	Pump2_Data_Exchange_Active_CMD_Value.16	:= GracoSealer_Inputs.Byte52.0;
	Pump2_Data_Exchange_Active_CMD_Value.17	:= GracoSealer_Inputs.Byte52.1;
	Pump2_Data_Exchange_Active_CMD_Value.18	:= GracoSealer_Inputs.Byte52.2;
	Pump2_Data_Exchange_Active_CMD_Value.19	:= GracoSealer_Inputs.Byte52.3;
	Pump2_Data_Exchange_Active_CMD_Value.20	:= GracoSealer_Inputs.Byte52.4;
	Pump2_Data_Exchange_Active_CMD_Value.21	:= GracoSealer_Inputs.Byte52.5;
	Pump2_Data_Exchange_Active_CMD_Value.22	:= GracoSealer_Inputs.Byte52.6;
	Pump2_Data_Exchange_Active_CMD_Value.23	:= GracoSealer_Inputs.Byte52.7;

	Pump2_Data_Exchange_Active_CMD_Value.24	:= GracoSealer_Inputs.Byte53.0;
	Pump2_Data_Exchange_Active_CMD_Value.25	:= GracoSealer_Inputs.Byte53.1;
	Pump2_Data_Exchange_Active_CMD_Value.26	:= GracoSealer_Inputs.Byte53.2;
	Pump2_Data_Exchange_Active_CMD_Value.27	:= GracoSealer_Inputs.Byte53.3;
	Pump2_Data_Exchange_Active_CMD_Value.28	:= GracoSealer_Inputs.Byte53.4;
	Pump2_Data_Exchange_Active_CMD_Value.29	:= GracoSealer_Inputs.Byte53.5;
	Pump2_Data_Exchange_Active_CMD_Value.30	:= GracoSealer_Inputs.Byte53.6;
	Pump2_Data_Exchange_Active_CMD_Value.31	:= GracoSealer_Inputs.Byte53.7;



	(*Heat 1 - Inputs from Graco*)
	Heat1_Heartbeat								:= GracoSealer_Inputs.Byte54.0;
	Heat1_Enabled								:= GracoSealer_Inputs.Byte54.1;
	Heat1_Control_Active							:= GracoSealer_Inputs.Byte54.2;
	Heat1_ON									:= GracoSealer_Inputs.Byte54.3;
	Heat1_WarmingUp							:= GracoSealer_Inputs.Byte54.4;
	Heat1_At_Temp								:= GracoSealer_Inputs.Byte54.5;
	Heat1_Temp_Soak_Mode						:= GracoSealer_Inputs.Byte54.6;
	Heat1_SetBack_Mode							:= GracoSealer_Inputs.Byte54.7;


	Heat1_Off									:= GracoSealer_Inputs.Byte55.0;
	Heat1_Module_NoAlarms_Active				:= GracoSealer_Inputs.Byte55.1;
	Heat1_Module_NoDeviations_Active				:= GracoSealer_Inputs.Byte55.2;
	Heat1_Module_NoAdvisory_Active				:= GracoSealer_Inputs.Byte55.3;
	Heat1_Zone_NoAlarms_Active					:= GracoSealer_Inputs.Byte55.4;
	Heat1_Zone_NoDeviations_Active				:= GracoSealer_Inputs.Byte55.5;
	Heat1_Zone_NoAdvisory_Active				:= GracoSealer_Inputs.Byte55.6;
	Heat1_Idle_Timeout_Happened					:= GracoSealer_Inputs.Byte55.7;


	(*Byte 56 Reserved*)
	(*Byte 57 Reserved*)


	Heat1_Soak_Time_Remaining.0					:= GracoSealer_Inputs.Byte58.0;			(*xx seconds*)
	Heat1_Soak_Time_Remaining.1					:= GracoSealer_Inputs.Byte58.1;			(*xx seconds*)
	Heat1_Soak_Time_Remaining.2					:= GracoSealer_Inputs.Byte58.2;			(*xx seconds*)
	Heat1_Soak_Time_Remaining.3					:= GracoSealer_Inputs.Byte58.3;			(*xx seconds*)
	Heat1_Soak_Time_Remaining.4					:= GracoSealer_Inputs.Byte58.4;			(*xx seconds*)
	Heat1_Soak_Time_Remaining.5					:= GracoSealer_Inputs.Byte58.5;			(*xx seconds*)
	Heat1_Soak_Time_Remaining.6					:= GracoSealer_Inputs.Byte58.6;			(*xx seconds*)
	Heat1_Soak_Time_Remaining.7					:= GracoSealer_Inputs.Byte58.7;			(*xx seconds*)

	Heat1_Soak_Time_Remaining.8					:= GracoSealer_Inputs.Byte59.0;			(*xx seconds*)
	Heat1_Soak_Time_Remaining.9					:= GracoSealer_Inputs.Byte59.1;			(*xx seconds*)
	Heat1_Soak_Time_Remaining.10				:= GracoSealer_Inputs.Byte59.2;			(*xx seconds*)
	Heat1_Soak_Time_Remaining.11				:= GracoSealer_Inputs.Byte59.3;			(*xx seconds*)
	Heat1_Soak_Time_Remaining.12				:= GracoSealer_Inputs.Byte59.4;			(*xx seconds*)
	Heat1_Soak_Time_Remaining.13				:= GracoSealer_Inputs.Byte59.5;			(*xx seconds*)
	Heat1_Soak_Time_Remaining.14				:= GracoSealer_Inputs.Byte59.6;			(*xx seconds*)
	Heat1_Soak_Time_Remaining.15				:= GracoSealer_Inputs.Byte59.7;			(*xx seconds*)


	Heat1_Data_Exchange_Active_CMD.0			:= GracoSealer_Inputs.Byte60.0;
	Heat1_Data_Exchange_Active_CMD.1			:= GracoSealer_Inputs.Byte60.1;
	Heat1_Data_Exchange_Active_CMD.2			:= GracoSealer_Inputs.Byte60.2;
	Heat1_Data_Exchange_Active_CMD.3			:= GracoSealer_Inputs.Byte60.3;
	Heat1_Data_Exchange_Active_CMD.4			:= GracoSealer_Inputs.Byte60.4;
	Heat1_Data_Exchange_Active_CMD.5			:= GracoSealer_Inputs.Byte60.5;
	Heat1_Data_Exchange_Active_CMD.6			:= GracoSealer_Inputs.Byte60.6;
	Heat1_Data_Exchange_Active_CMD.7			:= GracoSealer_Inputs.Byte60.7;

	Heat1_Data_Exchange_Active_CMD.8			:= GracoSealer_Inputs.Byte61.0;
	Heat1_Data_Exchange_Active_CMD.9			:= GracoSealer_Inputs.Byte61.1;
	Heat1_Data_Exchange_Active_CMD.10			:= GracoSealer_Inputs.Byte61.2;
	Heat1_Data_Exchange_Active_CMD.11			:= GracoSealer_Inputs.Byte61.3;
	Heat1_Data_Exchange_Active_CMD.12			:= GracoSealer_Inputs.Byte61.4;
	Heat1_Data_Exchange_Active_CMD.13			:= GracoSealer_Inputs.Byte61.5;
	Heat1_Data_Exchange_Active_CMD.14			:= GracoSealer_Inputs.Byte61.6;
	Heat1_Data_Exchange_Active_CMD.15			:= GracoSealer_Inputs.Byte61.7;


	Heat1_Data_Exchange_Active_CMD_Value.0		:= GracoSealer_Inputs.Byte62.0;
	Heat1_Data_Exchange_Active_CMD_Value.1		:= GracoSealer_Inputs.Byte62.1;
	Heat1_Data_Exchange_Active_CMD_Value.2		:= GracoSealer_Inputs.Byte62.2;
	Heat1_Data_Exchange_Active_CMD_Value.3		:= GracoSealer_Inputs.Byte62.3;
	Heat1_Data_Exchange_Active_CMD_Value.4		:= GracoSealer_Inputs.Byte62.4;
	Heat1_Data_Exchange_Active_CMD_Value.5		:= GracoSealer_Inputs.Byte62.5;
	Heat1_Data_Exchange_Active_CMD_Value.6		:= GracoSealer_Inputs.Byte62.6;
	Heat1_Data_Exchange_Active_CMD_Value.7		:= GracoSealer_Inputs.Byte62.7;

	Heat1_Data_Exchange_Active_CMD_Value.8		:= GracoSealer_Inputs.Byte63.0;
	Heat1_Data_Exchange_Active_CMD_Value.9		:= GracoSealer_Inputs.Byte63.1;
	Heat1_Data_Exchange_Active_CMD_Value.10		:= GracoSealer_Inputs.Byte63.2;
	Heat1_Data_Exchange_Active_CMD_Value.11		:= GracoSealer_Inputs.Byte63.3;
	Heat1_Data_Exchange_Active_CMD_Value.12		:= GracoSealer_Inputs.Byte63.4;
	Heat1_Data_Exchange_Active_CMD_Value.13		:= GracoSealer_Inputs.Byte63.5;
	Heat1_Data_Exchange_Active_CMD_Value.14		:= GracoSealer_Inputs.Byte63.6;
	Heat1_Data_Exchange_Active_CMD_Value.15		:= GracoSealer_Inputs.Byte63.7;

	Heat1_Data_Exchange_Active_CMD_Value.16		:= GracoSealer_Inputs.Byte64.0;
	Heat1_Data_Exchange_Active_CMD_Value.17		:= GracoSealer_Inputs.Byte64.1;
	Heat1_Data_Exchange_Active_CMD_Value.18		:= GracoSealer_Inputs.Byte64.2;
	Heat1_Data_Exchange_Active_CMD_Value.19		:= GracoSealer_Inputs.Byte64.3;
	Heat1_Data_Exchange_Active_CMD_Value.20		:= GracoSealer_Inputs.Byte64.4;
	Heat1_Data_Exchange_Active_CMD_Value.21		:= GracoSealer_Inputs.Byte64.5;
	Heat1_Data_Exchange_Active_CMD_Value.22		:= GracoSealer_Inputs.Byte64.6;
	Heat1_Data_Exchange_Active_CMD_Value.23		:= GracoSealer_Inputs.Byte64.7;

	Heat1_Data_Exchange_Active_CMD_Value.24		:= GracoSealer_Inputs.Byte65.0;
	Heat1_Data_Exchange_Active_CMD_Value.25		:= GracoSealer_Inputs.Byte65.1;
	Heat1_Data_Exchange_Active_CMD_Value.26		:= GracoSealer_Inputs.Byte65.2;
	Heat1_Data_Exchange_Active_CMD_Value.27		:= GracoSealer_Inputs.Byte65.3;
	Heat1_Data_Exchange_Active_CMD_Value.28		:= GracoSealer_Inputs.Byte65.4;
	Heat1_Data_Exchange_Active_CMD_Value.29		:= GracoSealer_Inputs.Byte65.5;
	Heat1_Data_Exchange_Active_CMD_Value.30		:= GracoSealer_Inputs.Byte65.6;
	Heat1_Data_Exchange_Active_CMD_Value.31		:= GracoSealer_Inputs.Byte65.7;



	(*Heat 2 - Inputs from Graco. Only used if tandem pump is on*)
	Heat1_Heartbeat								:= GracoSealer_Inputs.Byte66.0;
	Heat2_Enabled								:= GracoSealer_Inputs.Byte66.1;
	Heat2_Control_Active							:= GracoSealer_Inputs.Byte66.2;
	Heat2_ON									:= GracoSealer_Inputs.Byte66.3;
	Heat2_WarmingUp							:= GracoSealer_Inputs.Byte66.4;
	Heat2_At_Temp								:= GracoSealer_Inputs.Byte66.5;
	Heat2_Temp_Soak_Mode						:= GracoSealer_Inputs.Byte66.6;
	Heat2_SetBack_Mode							:= GracoSealer_Inputs.Byte66.7;


	Heat2_Off									:= GracoSealer_Inputs.Byte67.0;
	Heat2_Module_NoAlarms_Active				:= GracoSealer_Inputs.Byte67.1;
	Heat2_Module_NoDeviations_Active				:= GracoSealer_Inputs.Byte67.2;
	Heat2_Module_NoAdvisory_Active				:= GracoSealer_Inputs.Byte67.3;
	Heat2_Zone_NoAlarms_Active					:= GracoSealer_Inputs.Byte67.4;
	Heat2_Zone_NoDeviations_Active				:= GracoSealer_Inputs.Byte67.5;
	Heat2_Zone_NoAdvisory_Active				:= GracoSealer_Inputs.Byte67.6;
	Heat2_Idle_Timeout_Happened					:= GracoSealer_Inputs.Byte67.7;


	(*Byte 68 Reserved*)
	(*Byte 69 Reserved*)


	Heat2_Soak_Time_Remaining.0					:= GracoSealer_Inputs.Byte70.0;			(*xx seconds*)
	Heat2_Soak_Time_Remaining.1					:= GracoSealer_Inputs.Byte70.1;			(*xx seconds*)
	Heat2_Soak_Time_Remaining.2					:= GracoSealer_Inputs.Byte70.2;			(*xx seconds*)
	Heat2_Soak_Time_Remaining.3					:= GracoSealer_Inputs.Byte70.3;			(*xx seconds*)
	Heat2_Soak_Time_Remaining.4					:= GracoSealer_Inputs.Byte70.4;			(*xx seconds*)
	Heat2_Soak_Time_Remaining.5					:= GracoSealer_Inputs.Byte70.5;			(*xx seconds*)
	Heat2_Soak_Time_Remaining.6					:= GracoSealer_Inputs.Byte70.6;			(*xx seconds*)
	Heat2_Soak_Time_Remaining.7					:= GracoSealer_Inputs.Byte70.7;			(*xx seconds*)

	Heat2_Soak_Time_Remaining.8					:= GracoSealer_Inputs.Byte71.0;			(*xx seconds*)
	Heat2_Soak_Time_Remaining.9					:= GracoSealer_Inputs.Byte71.1;			(*xx seconds*)
	Heat2_Soak_Time_Remaining.10				:= GracoSealer_Inputs.Byte71.2;			(*xx seconds*)
	Heat2_Soak_Time_Remaining.11				:= GracoSealer_Inputs.Byte71.3;			(*xx seconds*)
	Heat2_Soak_Time_Remaining.12				:= GracoSealer_Inputs.Byte71.4;			(*xx seconds*)
	Heat2_Soak_Time_Remaining.13				:= GracoSealer_Inputs.Byte71.5;			(*xx seconds*)
	Heat2_Soak_Time_Remaining.14				:= GracoSealer_Inputs.Byte71.6;			(*xx seconds*)
	Heat2_Soak_Time_Remaining.15				:= GracoSealer_Inputs.Byte71.7;			(*xx seconds*)


	Heat2_Data_Exchange_Active_CMD.0			:= GracoSealer_Inputs.Byte72.0;
	Heat2_Data_Exchange_Active_CMD.1			:= GracoSealer_Inputs.Byte72.1;
	Heat2_Data_Exchange_Active_CMD.2			:= GracoSealer_Inputs.Byte72.2;
	Heat2_Data_Exchange_Active_CMD.3			:= GracoSealer_Inputs.Byte72.3;
	Heat2_Data_Exchange_Active_CMD.4			:= GracoSealer_Inputs.Byte72.4;
	Heat2_Data_Exchange_Active_CMD.5			:= GracoSealer_Inputs.Byte72.5;
	Heat2_Data_Exchange_Active_CMD.6			:= GracoSealer_Inputs.Byte72.6;
	Heat2_Data_Exchange_Active_CMD.7			:= GracoSealer_Inputs.Byte72.7;

	Heat2_Data_Exchange_Active_CMD.8			:= GracoSealer_Inputs.Byte73.0;
	Heat2_Data_Exchange_Active_CMD.9			:= GracoSealer_Inputs.Byte73.1;
	Heat2_Data_Exchange_Active_CMD.10			:= GracoSealer_Inputs.Byte73.2;
	Heat2_Data_Exchange_Active_CMD.11			:= GracoSealer_Inputs.Byte73.3;
	Heat2_Data_Exchange_Active_CMD.12			:= GracoSealer_Inputs.Byte73.4;
	Heat2_Data_Exchange_Active_CMD.13			:= GracoSealer_Inputs.Byte73.5;
	Heat2_Data_Exchange_Active_CMD.14			:= GracoSealer_Inputs.Byte73.6;
	Heat2_Data_Exchange_Active_CMD.15			:= GracoSealer_Inputs.Byte73.7;


	Heat2_Data_Exchange_Active_CMD_Value.0		:= GracoSealer_Inputs.Byte74.0;
	Heat2_Data_Exchange_Active_CMD_Value.1		:= GracoSealer_Inputs.Byte74.1;
	Heat2_Data_Exchange_Active_CMD_Value.2		:= GracoSealer_Inputs.Byte74.2;
	Heat2_Data_Exchange_Active_CMD_Value.3		:= GracoSealer_Inputs.Byte74.3;
	Heat2_Data_Exchange_Active_CMD_Value.4		:= GracoSealer_Inputs.Byte74.4;
	Heat2_Data_Exchange_Active_CMD_Value.5		:= GracoSealer_Inputs.Byte74.5;
	Heat2_Data_Exchange_Active_CMD_Value.6		:= GracoSealer_Inputs.Byte74.6;
	Heat2_Data_Exchange_Active_CMD_Value.7		:= GracoSealer_Inputs.Byte74.7;

	Heat2_Data_Exchange_Active_CMD_Value.8		:= GracoSealer_Inputs.Byte75.0;
	Heat2_Data_Exchange_Active_CMD_Value.9		:= GracoSealer_Inputs.Byte75.1;
	Heat2_Data_Exchange_Active_CMD_Value.10		:= GracoSealer_Inputs.Byte75.2;
	Heat2_Data_Exchange_Active_CMD_Value.11		:= GracoSealer_Inputs.Byte75.3;
	Heat2_Data_Exchange_Active_CMD_Value.12		:= GracoSealer_Inputs.Byte75.4;
	Heat2_Data_Exchange_Active_CMD_Value.13		:= GracoSealer_Inputs.Byte75.5;
	Heat2_Data_Exchange_Active_CMD_Value.14		:= GracoSealer_Inputs.Byte75.6;
	Heat2_Data_Exchange_Active_CMD_Value.15		:= GracoSealer_Inputs.Byte75.7;

	Heat2_Data_Exchange_Active_CMD_Value.16		:= GracoSealer_Inputs.Byte76.0;
	Heat2_Data_Exchange_Active_CMD_Value.17		:= GracoSealer_Inputs.Byte76.1;
	Heat2_Data_Exchange_Active_CMD_Value.18		:= GracoSealer_Inputs.Byte76.2;
	Heat2_Data_Exchange_Active_CMD_Value.19		:= GracoSealer_Inputs.Byte76.3;
	Heat2_Data_Exchange_Active_CMD_Value.20		:= GracoSealer_Inputs.Byte76.4;
	Heat2_Data_Exchange_Active_CMD_Value.21		:= GracoSealer_Inputs.Byte76.5;
	Heat2_Data_Exchange_Active_CMD_Value.22		:= GracoSealer_Inputs.Byte76.6;
	Heat2_Data_Exchange_Active_CMD_Value.23		:= GracoSealer_Inputs.Byte76.7;

	Heat2_Data_Exchange_Active_CMD_Value.24		:= GracoSealer_Inputs.Byte77.0;
	Heat2_Data_Exchange_Active_CMD_Value.25		:= GracoSealer_Inputs.Byte77.1;
	Heat2_Data_Exchange_Active_CMD_Value.26		:= GracoSealer_Inputs.Byte77.2;
	Heat2_Data_Exchange_Active_CMD_Value.27		:= GracoSealer_Inputs.Byte77.3;
	Heat2_Data_Exchange_Active_CMD_Value.28		:= GracoSealer_Inputs.Byte77.4;
	Heat2_Data_Exchange_Active_CMD_Value.29		:= GracoSealer_Inputs.Byte77.5;
	Heat2_Data_Exchange_Active_CMD_Value.30		:= GracoSealer_Inputs.Byte77.6;
	Heat2_Data_Exchange_Active_CMD_Value.31		:= GracoSealer_Inputs.Byte77.7;







































(*end*)
END_ACTION

ACTION Outputs:



	GracoSealer_Outputs.Byte0.0	:= Pump1_Sys_Data_Exchange_CMD.0;
	GracoSealer_Outputs.Byte0.1	:= Pump1_Sys_Data_Exchange_CMD.1;
	GracoSealer_Outputs.Byte0.2	:= Pump1_Sys_Data_Exchange_CMD.2;
	GracoSealer_Outputs.Byte0.3	:= Pump1_Sys_Data_Exchange_CMD.3;
	GracoSealer_Outputs.Byte0.4	:= Pump1_Sys_Data_Exchange_CMD.4;
	GracoSealer_Outputs.Byte0.5	:= Pump1_Sys_Data_Exchange_CMD.5;
	GracoSealer_Outputs.Byte0.6	:= Pump1_Sys_Data_Exchange_CMD.6;
	GracoSealer_Outputs.Byte0.7	:= Pump1_Sys_Data_Exchange_CMD.7;

	GracoSealer_Outputs.Byte1.0	:= Pump1_Sys_Data_Exchange_CMD.8;
	GracoSealer_Outputs.Byte1.1	:= Pump1_Sys_Data_Exchange_CMD.9;
	GracoSealer_Outputs.Byte1.2	:= Pump1_Sys_Data_Exchange_CMD.10;
	GracoSealer_Outputs.Byte1.3	:= Pump1_Sys_Data_Exchange_CMD.11;
	GracoSealer_Outputs.Byte1.4	:= Pump1_Sys_Data_Exchange_CMD.12;
	GracoSealer_Outputs.Byte1.5	:= Pump1_Sys_Data_Exchange_CMD.13;
	GracoSealer_Outputs.Byte1.6	:= Pump1_Sys_Data_Exchange_CMD.14;
	GracoSealer_Outputs.Byte1.7	:= Pump1_Sys_Data_Exchange_CMD.15;


	GracoSealer_Outputs.Byte2.0	:= Pump1_Sys_Enable;
	GracoSealer_Outputs.Byte2.1	:= Pump1_Sys_Disable_REQ;
	GracoSealer_Outputs.Byte2.2	:= Pump1_Lockout;
	GracoSealer_Outputs.Byte2.3	:= Pump1_Style_Enable;
	GracoSealer_Outputs.Byte2.4	:= Pump1_Go;
	GracoSealer_Outputs.Byte2.5	:= Pump1_Disp_Complete;
	GracoSealer_Outputs.Byte2.6	:= Pump1_Tandem_Cross_REQ;
	GracoSealer_Outputs.Byte2.7	:= Pump2_Prime_Inactive_Pump_REQ;


	GracoSealer_Outputs.Byte3.0	:= Pump1_Valve_Depressurization_REQ;
	GracoSealer_Outputs.Byte3.1	:= Pump1_Platen_Depressurization_REQ;
	GracoSealer_Outputs.Byte3.2	:= Pump1_Auto_Depressurization_Cancel_REQ;
	GracoSealer_Outputs.Byte3.3	:= Pump_Acknowledge_Clear_Errors;
	(*Byte3.4 Reserved Bit 1*)
	(*Byte3.5 Reserved Bit 2*)
	(*Byte 3.6 Reserved Bit 3*)
	(*Byte 3.7 Reserved Bit 4*)


	GracoSealer_Outputs.Byte4.0	:= Pump1_Desired_Style_Numb.0;
	GracoSealer_Outputs.Byte4.1	:= Pump1_Desired_Style_Numb.1;
	GracoSealer_Outputs.Byte4.2	:= Pump1_Desired_Style_Numb.2;
	GracoSealer_Outputs.Byte4.3	:= Pump1_Desired_Style_Numb.3;
	GracoSealer_Outputs.Byte4.4	:= Pump1_Desired_Style_Numb.4;
	GracoSealer_Outputs.Byte4.5	:= Pump1_Desired_Style_Numb.5;
	GracoSealer_Outputs.Byte4.6	:= Pump1_Desired_Style_Numb.6;
	GracoSealer_Outputs.Byte4.7	:= Pump1_Desired_Style_Numb.7;

	GracoSealer_Outputs.Byte5.0	:= Pump1_Desired_Style_Numb.8;
	GracoSealer_Outputs.Byte5.1	:= Pump1_Desired_Style_Numb.9;
	GracoSealer_Outputs.Byte5.2	:= Pump1_Desired_Style_Numb.10;
	GracoSealer_Outputs.Byte5.3	:= Pump1_Desired_Style_Numb.11;
	GracoSealer_Outputs.Byte5.4	:= Pump1_Desired_Style_Numb.12;
	GracoSealer_Outputs.Byte5.5	:= Pump1_Desired_Style_Numb.13;
	GracoSealer_Outputs.Byte5.6	:= Pump1_Desired_Style_Numb.14;
	GracoSealer_Outputs.Byte5.7	:= Pump1_Desired_Style_Numb.15;


	GracoSealer_Outputs.Byte6.0	:= Pump1_Style_PreCharge_REQ.0;		(*xxx.x bars*)
	GracoSealer_Outputs.Byte6.1	:= Pump1_Style_PreCharge_REQ.1;		(*xxx.x bars*)
	GracoSealer_Outputs.Byte6.2	:= Pump1_Style_PreCharge_REQ.2;		(*xxx.x bars*)
	GracoSealer_Outputs.Byte6.3	:= Pump1_Style_PreCharge_REQ.3;		(*xxx.x bars*)
	GracoSealer_Outputs.Byte6.4	:= Pump1_Style_PreCharge_REQ.4;		(*xxx.x bars*)
	GracoSealer_Outputs.Byte6.5	:= Pump1_Style_PreCharge_REQ.5;		(*xxx.x bars*)
	GracoSealer_Outputs.Byte6.6	:= Pump1_Style_PreCharge_REQ.6;		(*xxx.x bars*)
	GracoSealer_Outputs.Byte6.7	:= Pump1_Style_PreCharge_REQ.7;		(*xxx.x bars*)

	GracoSealer_Outputs.Byte7.0	:= Pump1_Style_PreCharge_REQ.8;		(*xxx.x bars*)
	GracoSealer_Outputs.Byte7.1	:= Pump1_Style_PreCharge_REQ.9;		(*xxx.x bars*)
	GracoSealer_Outputs.Byte7.2	:= Pump1_Style_PreCharge_REQ.10;		(*xxx.x bars*)
	GracoSealer_Outputs.Byte7.3	:= Pump1_Style_PreCharge_REQ.11;		(*xxx.x bars*)
	GracoSealer_Outputs.Byte7.4	:= Pump1_Style_PreCharge_REQ.12;		(*xxx.x bars*)
	GracoSealer_Outputs.Byte7.5	:= Pump1_Style_PreCharge_REQ.13;		(*xxx.x bars*)
	GracoSealer_Outputs.Byte7.6	:= Pump1_Style_PreCharge_REQ.14;		(*xxx.x bars*)
	GracoSealer_Outputs.Byte7.7	:= Pump1_Style_PreCharge_REQ.15;		(*xxx.x bars*)


	GracoSealer_Outputs.Byte8.0	:= Pump1_FlowRate_REQ.0;			(*xxxx cc/min*)
	GracoSealer_Outputs.Byte8.1	:= Pump1_FlowRate_REQ.1;			(*xxxx cc/min*)
	GracoSealer_Outputs.Byte8.2	:= Pump1_FlowRate_REQ.2;			(*xxxx cc/min*)
	GracoSealer_Outputs.Byte8.3	:= Pump1_FlowRate_REQ.3;			(*xxxx cc/min*)
	GracoSealer_Outputs.Byte8.4	:= Pump1_FlowRate_REQ.4;			(*xxxx cc/min*)
	GracoSealer_Outputs.Byte8.5	:= Pump1_FlowRate_REQ.5;			(*xxxx cc/min*)
	GracoSealer_Outputs.Byte8.6	:= Pump1_FlowRate_REQ.6;			(*xxxx cc/min*)
	GracoSealer_Outputs.Byte8.7	:= Pump1_FlowRate_REQ.7;			(*xxxx cc/min*)

	GracoSealer_Outputs.Byte9.0	:= Pump1_FlowRate_REQ.8;			(*xxxx cc/min*)
	GracoSealer_Outputs.Byte9.1	:= Pump1_FlowRate_REQ.9;			(*xxxx cc/min*)
	GracoSealer_Outputs.Byte9.2	:= Pump1_FlowRate_REQ.10;			(*xxxx cc/min*)
	GracoSealer_Outputs.Byte9.3	:= Pump1_FlowRate_REQ.11;			(*xxxx cc/min*)
	GracoSealer_Outputs.Byte9.4	:= Pump1_FlowRate_REQ.12;			(*xxxx cc/min*)
	GracoSealer_Outputs.Byte9.5	:= Pump1_FlowRate_REQ.13;			(*xxxx cc/min*)
	GracoSealer_Outputs.Byte9.6	:= Pump1_FlowRate_REQ.14;			(*xxxx cc/min*)
	GracoSealer_Outputs.Byte9.7	:= Pump1_FlowRate_REQ.15;			(*xxxx cc/min*)


	GracoSealer_Outputs.Byte10.0	:= Pump1_ShotSize_REQ.0;				(*xxx.xx cc*)
	GracoSealer_Outputs.Byte10.1	:= Pump1_ShotSize_REQ.1;				(*xxx.xx cc*)
	GracoSealer_Outputs.Byte10.2	:= Pump1_ShotSize_REQ.2;				(*xxx.xx cc*)
	GracoSealer_Outputs.Byte10.3	:= Pump1_ShotSize_REQ.3;				(*xxx.xx cc*)
	GracoSealer_Outputs.Byte10.4	:= Pump1_ShotSize_REQ.4;				(*xxx.xx cc*)
	GracoSealer_Outputs.Byte10.5	:= Pump1_ShotSize_REQ.5;				(*xxx.xx cc*)
	GracoSealer_Outputs.Byte10.6	:= Pump1_ShotSize_REQ.6;				(*xxx.xx cc*)
	GracoSealer_Outputs.Byte10.7	:= Pump1_ShotSize_REQ.7;				(*xxx.xx cc*)

	GracoSealer_Outputs.Byte11.0	:= Pump1_ShotSize_REQ.8;				(*xxx.xx cc*)
	GracoSealer_Outputs.Byte11.1	:= Pump1_ShotSize_REQ.9;				(*xxx.xx cc*)
	GracoSealer_Outputs.Byte11.2	:= Pump1_ShotSize_REQ.10;			(*xxx.xx cc*)
	GracoSealer_Outputs.Byte11.3	:= Pump1_ShotSize_REQ.11;			(*xxx.xx cc*)
	GracoSealer_Outputs.Byte11.4	:= Pump1_ShotSize_REQ.12;			(*xxx.xx cc*)
	GracoSealer_Outputs.Byte11.5	:= Pump1_ShotSize_REQ.13;			(*xxx.xx cc*)
	GracoSealer_Outputs.Byte11.6	:= Pump1_ShotSize_REQ.14;			(*xxx.xx cc*)
	GracoSealer_Outputs.Byte11.7	:= Pump1_ShotSize_REQ.15;			(*xxx.xx cc*)


	GracoSealer_Outputs.Byte12.0	:= Pump2_PrimePressure_Target.0;		(*xxx.x bars*)
	GracoSealer_Outputs.Byte12.1	:= Pump2_PrimePressure_Target.1;		(*xxx.x bars*)
	GracoSealer_Outputs.Byte12.2	:= Pump2_PrimePressure_Target.2;		(*xxx.x bars*)
	GracoSealer_Outputs.Byte12.3	:= Pump2_PrimePressure_Target.3;		(*xxx.x bars*)
	GracoSealer_Outputs.Byte12.4	:= Pump2_PrimePressure_Target.4;		(*xxx.x bars*)
	GracoSealer_Outputs.Byte12.5	:= Pump2_PrimePressure_Target.5;		(*xxx.x bars*)
	GracoSealer_Outputs.Byte12.6	:= Pump2_PrimePressure_Target.6;		(*xxx.x bars*)
	GracoSealer_Outputs.Byte12.7	:= Pump2_PrimePressure_Target.7;		(*xxx.x bars*)

	GracoSealer_Outputs.Byte13.0	:= Pump2_PrimePressure_Target.8;		(*xxx.x bars*)
	GracoSealer_Outputs.Byte13.1	:= Pump2_PrimePressure_Target.9;		(*xxx.x bars*)
	GracoSealer_Outputs.Byte13.2	:= Pump2_PrimePressure_Target.10;		(*xxx.x bars*)
	GracoSealer_Outputs.Byte13.3	:= Pump2_PrimePressure_Target.11;		(*xxx.x bars*)
	GracoSealer_Outputs.Byte13.4	:= Pump2_PrimePressure_Target.12;		(*xxx.x bars*)
	GracoSealer_Outputs.Byte13.5	:= Pump2_PrimePressure_Target.13;		(*xxx.x bars*)
	GracoSealer_Outputs.Byte13.6	:= Pump2_PrimePressure_Target.14;		(*xxx.x bars*)
	GracoSealer_Outputs.Byte13.7	:= Pump2_PrimePressure_Target.15;		(*xxx.x bars*)


	GracoSealer_Outputs.Byte14.0	:= Pump2_PrimeFlow_Target.0;			(*xxxx cc/min*)
	GracoSealer_Outputs.Byte14.1	:= Pump2_PrimeFlow_Target.1;			(*xxxx cc/min*)
	GracoSealer_Outputs.Byte14.2	:= Pump2_PrimeFlow_Target.2;			(*xxxx cc/min*)
	GracoSealer_Outputs.Byte14.3	:= Pump2_PrimeFlow_Target.3;			(*xxxx cc/min*)
	GracoSealer_Outputs.Byte14.4	:= Pump2_PrimeFlow_Target.4;			(*xxxx cc/min*)
	GracoSealer_Outputs.Byte14.5	:= Pump2_PrimeFlow_Target.5;			(*xxxx cc/min*)
	GracoSealer_Outputs.Byte14.6	:= Pump2_PrimeFlow_Target.6;			(*xxxx cc/min*)
	GracoSealer_Outputs.Byte14.7	:= Pump2_PrimeFlow_Target.7;			(*xxxx cc/min*)

	GracoSealer_Outputs.Byte15.0	:= Pump2_PrimeFlow_Target.8;			(*xxxx cc/min*)
	GracoSealer_Outputs.Byte15.1	:= Pump2_PrimeFlow_Target.9;			(*xxxx cc/min*)
	GracoSealer_Outputs.Byte15.2	:= Pump2_PrimeFlow_Target.10;			(*xxxx cc/min*)
	GracoSealer_Outputs.Byte15.3	:= Pump2_PrimeFlow_Target.11;			(*xxxx cc/min*)
	GracoSealer_Outputs.Byte15.4	:= Pump2_PrimeFlow_Target.12;			(*xxxx cc/min*)
	GracoSealer_Outputs.Byte15.5	:= Pump2_PrimeFlow_Target.13;			(*xxxx cc/min*)
	GracoSealer_Outputs.Byte15.6	:= Pump2_PrimeFlow_Target.14;			(*xxxx cc/min*)
	GracoSealer_Outputs.Byte15.7	:= Pump2_PrimeFlow_Target.15;			(*xxxx cc/min*)


	GracoSealer_Outputs.Byte16.0	:= Heat1_HeatEnabled_REQ;
	GracoSealer_Outputs.Byte16.1	:= Heat1_HeatDissabled_REQ;
	GracoSealer_Outputs.Byte16.2	:= Heat1_PLC_Lockout;
	GracoSealer_Outputs.Byte16.3	:= Heat1_Heat_ON_REQ;
	GracoSealer_Outputs.Byte16.4	:= Heat1_Heat_OFF_REQ;
	GracoSealer_Outputs.Byte16.5	:= Heat1_Setback_REQ;
	GracoSealer_Outputs.Byte16.6	:= Heat1_Acknowledge_Clear_Errors;
	(*Byte 16.7 Reserved Bit 1*)


	(*Byte 17 Reserved*)


	GracoSealer_Outputs.Byte18.0	:= Heat1_Data_Exchange_CMD.0;
	GracoSealer_Outputs.Byte18.1	:= Heat1_Data_Exchange_CMD.1;
	GracoSealer_Outputs.Byte18.2	:= Heat1_Data_Exchange_CMD.2;
	GracoSealer_Outputs.Byte18.3	:= Heat1_Data_Exchange_CMD.3;
	GracoSealer_Outputs.Byte18.4	:= Heat1_Data_Exchange_CMD.4;
	GracoSealer_Outputs.Byte18.5	:= Heat1_Data_Exchange_CMD.5;
	GracoSealer_Outputs.Byte18.6	:= Heat1_Data_Exchange_CMD.6;
	GracoSealer_Outputs.Byte18.7	:= Heat1_Data_Exchange_CMD.7;

	GracoSealer_Outputs.Byte19.0	:= Heat1_Data_Exchange_CMD.8;
	GracoSealer_Outputs.Byte19.1	:= Heat1_Data_Exchange_CMD.9;
	GracoSealer_Outputs.Byte19.2	:= Heat1_Data_Exchange_CMD.10;
	GracoSealer_Outputs.Byte19.3	:= Heat1_Data_Exchange_CMD.11;
	GracoSealer_Outputs.Byte19.4	:= Heat1_Data_Exchange_CMD.12;
	GracoSealer_Outputs.Byte19.5	:= Heat1_Data_Exchange_CMD.13;
	GracoSealer_Outputs.Byte19.6	:= Heat1_Data_Exchange_CMD.14;
	GracoSealer_Outputs.Byte19.7	:= Heat1_Data_Exchange_CMD.15;

	GracoSealer_Outputs.Byte20.0	:= Heat1_Data_Exchange_CMD_Value.0;
	GracoSealer_Outputs.Byte20.1	:= Heat1_Data_Exchange_CMD_Value.1;
	GracoSealer_Outputs.Byte20.2	:= Heat1_Data_Exchange_CMD_Value.2;
	GracoSealer_Outputs.Byte20.3	:= Heat1_Data_Exchange_CMD_Value.3;
	GracoSealer_Outputs.Byte20.4	:= Heat1_Data_Exchange_CMD_Value.4;
	GracoSealer_Outputs.Byte20.5	:= Heat1_Data_Exchange_CMD_Value.5;
	GracoSealer_Outputs.Byte20.6	:= Heat1_Data_Exchange_CMD_Value.6;
	GracoSealer_Outputs.Byte20.7	:= Heat1_Data_Exchange_CMD_Value.7;

	GracoSealer_Outputs.Byte21.0	:= Heat1_Data_Exchange_CMD_Value.8;
	GracoSealer_Outputs.Byte21.1	:= Heat1_Data_Exchange_CMD_Value.9;
	GracoSealer_Outputs.Byte21.2	:= Heat1_Data_Exchange_CMD_Value.10;
	GracoSealer_Outputs.Byte21.3	:= Heat1_Data_Exchange_CMD_Value.11;
	GracoSealer_Outputs.Byte21.4	:= Heat1_Data_Exchange_CMD_Value.12;
	GracoSealer_Outputs.Byte21.5	:= Heat1_Data_Exchange_CMD_Value.13;
	GracoSealer_Outputs.Byte21.6	:= Heat1_Data_Exchange_CMD_Value.14;
	GracoSealer_Outputs.Byte21.7	:= Heat1_Data_Exchange_CMD_Value.15;

	GracoSealer_Outputs.Byte22.0	:= Heat1_Data_Exchange_CMD_Value.16;
	GracoSealer_Outputs.Byte22.1	:= Heat1_Data_Exchange_CMD_Value.17;
	GracoSealer_Outputs.Byte22.2	:= Heat1_Data_Exchange_CMD_Value.18;
	GracoSealer_Outputs.Byte22.3	:= Heat1_Data_Exchange_CMD_Value.19;
	GracoSealer_Outputs.Byte22.4	:= Heat1_Data_Exchange_CMD_Value.20;
	GracoSealer_Outputs.Byte22.5	:= Heat1_Data_Exchange_CMD_Value.21;
	GracoSealer_Outputs.Byte22.6	:= Heat1_Data_Exchange_CMD_Value.22;
	GracoSealer_Outputs.Byte22.7	:= Heat1_Data_Exchange_CMD_Value.23;

	GracoSealer_Outputs.Byte23.0	:= Heat1_Data_Exchange_CMD_Value.24;
	GracoSealer_Outputs.Byte23.1	:= Heat1_Data_Exchange_CMD_Value.25;
	GracoSealer_Outputs.Byte23.2	:= Heat1_Data_Exchange_CMD_Value.26;
	GracoSealer_Outputs.Byte23.3	:= Heat1_Data_Exchange_CMD_Value.27;
	GracoSealer_Outputs.Byte23.4	:= Heat1_Data_Exchange_CMD_Value.28;
	GracoSealer_Outputs.Byte23.5	:= Heat1_Data_Exchange_CMD_Value.29;
	GracoSealer_Outputs.Byte23.6	:= Heat1_Data_Exchange_CMD_Value.30;
	GracoSealer_Outputs.Byte23.7	:= Heat1_Data_Exchange_CMD_Value.31;


	GracoSealer_Outputs.Byte24.0	:= Heat2_HeatEnabled_REQ;
	GracoSealer_Outputs.Byte24.1	:= Heat2_HeatDissabled_REQ;
	GracoSealer_Outputs.Byte24.2	:= Heat2_PLC_Lockout;
	GracoSealer_Outputs.Byte24.3	:= Heat2_Heat_ON_REQ;
	GracoSealer_Outputs.Byte24.4	:= Heat2_Heat_OFF_REQ;
	GracoSealer_Outputs.Byte24.5	:= Heat2_Setback_REQ;
	GracoSealer_Outputs.Byte24.6	:= Heat2_Acknowledge_Clear_Errors;
	(*Byte 24.7 Reserved Bit 1*)


	(*Byte 25 Reserved*)


	GracoSealer_Outputs.Byte26.0	:= Heat2_Data_Exchange_CMD.0;
	GracoSealer_Outputs.Byte26.1	:= Heat2_Data_Exchange_CMD.1;
	GracoSealer_Outputs.Byte26.2	:= Heat2_Data_Exchange_CMD.2;
	GracoSealer_Outputs.Byte26.3	:= Heat2_Data_Exchange_CMD.3;
	GracoSealer_Outputs.Byte26.4	:= Heat2_Data_Exchange_CMD.4;
	GracoSealer_Outputs.Byte26.5	:= Heat2_Data_Exchange_CMD.5;
	GracoSealer_Outputs.Byte26.6	:= Heat2_Data_Exchange_CMD.6;
	GracoSealer_Outputs.Byte26.7	:= Heat2_Data_Exchange_CMD.7;

	GracoSealer_Outputs.Byte27.0	:= Heat2_Data_Exchange_CMD.8;
	GracoSealer_Outputs.Byte27.1	:= Heat2_Data_Exchange_CMD.9;
	GracoSealer_Outputs.Byte27.2	:= Heat2_Data_Exchange_CMD.10;
	GracoSealer_Outputs.Byte27.3	:= Heat2_Data_Exchange_CMD.11;
	GracoSealer_Outputs.Byte27.4	:= Heat2_Data_Exchange_CMD.12;
	GracoSealer_Outputs.Byte27.5	:= Heat2_Data_Exchange_CMD.13;
	GracoSealer_Outputs.Byte27.6	:= Heat2_Data_Exchange_CMD.14;
	GracoSealer_Outputs.Byte27.7	:= Heat2_Data_Exchange_CMD.15;


	GracoSealer_Outputs.Byte28.0	:= Heat2_Data_Exchange_CMD_Value.0;
	GracoSealer_Outputs.Byte28.1	:= Heat2_Data_Exchange_CMD_Value.1;
	GracoSealer_Outputs.Byte28.2	:= Heat2_Data_Exchange_CMD_Value.2;
	GracoSealer_Outputs.Byte28.3	:= Heat2_Data_Exchange_CMD_Value.3;
	GracoSealer_Outputs.Byte28.4	:= Heat2_Data_Exchange_CMD_Value.4;
	GracoSealer_Outputs.Byte28.5	:= Heat2_Data_Exchange_CMD_Value.5;
	GracoSealer_Outputs.Byte28.6	:= Heat2_Data_Exchange_CMD_Value.6;
	GracoSealer_Outputs.Byte28.7	:= Heat2_Data_Exchange_CMD_Value.7;

	GracoSealer_Outputs.Byte29.0	:= Heat2_Data_Exchange_CMD_Value.8;
	GracoSealer_Outputs.Byte29.1	:= Heat2_Data_Exchange_CMD_Value.9;
	GracoSealer_Outputs.Byte29.2	:= Heat2_Data_Exchange_CMD_Value.10;
	GracoSealer_Outputs.Byte29.3	:= Heat2_Data_Exchange_CMD_Value.11;
	GracoSealer_Outputs.Byte29.4	:= Heat2_Data_Exchange_CMD_Value.12;
	GracoSealer_Outputs.Byte29.5	:= Heat2_Data_Exchange_CMD_Value.13;
	GracoSealer_Outputs.Byte29.6	:= Heat2_Data_Exchange_CMD_Value.14;
	GracoSealer_Outputs.Byte29.7	:= Heat2_Data_Exchange_CMD_Value.15;

	GracoSealer_Outputs.Byte30.0	:= Heat2_Data_Exchange_CMD_Value.16;
	GracoSealer_Outputs.Byte30.1	:= Heat2_Data_Exchange_CMD_Value.17;
	GracoSealer_Outputs.Byte30.2	:= Heat2_Data_Exchange_CMD_Value.18;
	GracoSealer_Outputs.Byte30.3	:= Heat2_Data_Exchange_CMD_Value.19;
	GracoSealer_Outputs.Byte30.4	:= Heat2_Data_Exchange_CMD_Value.20;
	GracoSealer_Outputs.Byte30.5	:= Heat2_Data_Exchange_CMD_Value.21;
	GracoSealer_Outputs.Byte30.6	:= Heat2_Data_Exchange_CMD_Value.22;
	GracoSealer_Outputs.Byte30.7	:= Heat2_Data_Exchange_CMD_Value.23;

	GracoSealer_Outputs.Byte31.0	:= Heat2_Data_Exchange_CMD_Value.24;
	GracoSealer_Outputs.Byte31.1	:= Heat2_Data_Exchange_CMD_Value.25;
	GracoSealer_Outputs.Byte31.2	:= Heat2_Data_Exchange_CMD_Value.26;
	GracoSealer_Outputs.Byte31.3	:= Heat2_Data_Exchange_CMD_Value.27;
	GracoSealer_Outputs.Byte31.4	:= Heat2_Data_Exchange_CMD_Value.28;
	GracoSealer_Outputs.Byte31.5	:= Heat2_Data_Exchange_CMD_Value.29;
	GracoSealer_Outputs.Byte31.6	:= Heat2_Data_Exchange_CMD_Value.30;
	GracoSealer_Outputs.Byte31.7	:= Heat2_Data_Exchange_CMD_Value.31;
































(*end*)
END_ACTION

END_FUNCTION_BLOCK

// ---- POUs/FBs/FB_GTAC_NutWeldLVDT_20250612.TcPOU
(*FB for use with Vision Nutwelders

	Original Author(s): Jessy Underhill of Sodecia GTAC.; 
------------------------------------------------------------------------------------------
REVISION NOTES:
	Version 20210216
		- intial concept, j.underhill
	Version 20250612
		- Eliminated hard typed M6/M8 code and reduced to singular generic LVDT functionality, b.lekx-toniolo
------------------------------------------------------------------------------------------
*)

FUNCTION_BLOCK FB_GTAC_NutWeldLVDT_20250612
VAR_INPUT

	Model_ID: UDINT;								(*Model ID Input from Fixture*)
	Option_InScaledValues: BOOL;							(*True = Used Sclaed LVDT Values, False = use Raw LVDT Values*)
	Save_LVDT_Conf: BOOL;							(*Input from UI to Save LVDT Values*)
	Save_Nut_Conf: BOOL;							(*Input from UI to Save Nut Values*)

	Raw_Transducer: REAL;						(*Scaled Value from Transducer EL3255 Channel*)

	Ready_For_Measurement: BOOL;				(*Weld Gun Reached Force - Ready to Measure Transducer/LVDT*)
	Weld_Complete: BOOL;							(*Used to Reset Nut Orientation OK AFTER Weld Complete*)
	Reset_NutOK: BOOL;							(*Used to Clear NutOK Bits in Case that Weld Complete is not acheived*)


	NutInput_UpperLimit: ARRAY [0..40] OF REAL;	(*Input from UI to adjust the transducer upper limits for each Model*)
	NutInput_LowerLimit: ARRAY [0..40] OF REAL;	(*Input from UI to adjust the transducer lower limits for each Model*)

END_VAR

VAR PERSISTENT

	Nut_UpperLimit: ARRAY [0..40] OF REAL;		(*Array for storing the Upper Limits for Nut Orientation, for each model*)
	Nut_LowerLimit: ARRAY [0..40] OF REAL;		(*Array for storing the Lower Limits for Nut Orientation, for each model*)

	Last_Nut_Raw: UINT;

END_VAR

VAR
	FB_OK: BOOL;

	Trig_NutLVDT: R_TRIG;

	Weld_Dwell: TON;
	LVDT_Scaled: REAL;
	
	Store: R_TRIG;

	NutWeld_Store: ARRAY [0..50] OF REAL;	(*Store Last 50 LVDT Measurements for Welds*)

END_VAR

VAR_OUTPUT

	LVDT_Saved: BOOL;			(*Indicates LVDT Values have been properly saved from HMI settings into PLC*)

	NutPrev_Scaled: REAL;					(*Store the Last LVDT Sclaed Measurement for Nut Weld*)
	NutPrev_Raw: REAL;					(*Store the Last LVDT Raw Measurement for Nut Weld*)

	NutOK: BOOL;				(*Capture M6 Nut OK for all part models*)

END_VAR

FB_OK:= TRUE;

	(*LVDT Scaling*)
	LVDT_Scaled:= FUN_GTAC_Scaling(
						Raw_Transducer,					(*Raw Data to Scale*)
						3570,							(*Unscaled Lower Limit - JAU, WAS 2170, then 12800, then 3800, then 11200, then 3570*)
						15400,							(*Unscaled Upper Limit - JAU, WAS 14250, then 23000, then 16200, then 21550, then 15400*)
						0, 								(*Scaled Lower Limit - Pin RETD*)
						22								(*Scaled Upper Limit - Pin ADVD*)
						);




	(*Save LVDT Limits from HMI User Input*)
	IF Save_LVDT_Conf
		THEN
			(*Nut Present - upper limit*)
			Nut_UpperLimit[Model_ID]:= NutInput_UpperLimit[Model_ID];
			(*Nut Present - lower limit*)
			Nut_LowerLimit[Model_ID]:= NutInput_LowerLimit[Model_ID];
	END_IF;

	(*Weld Dwell - Wait for Nut Measurment to Settle*)
	Weld_Dwell.IN:= Ready_For_Measurement;
	Weld_Dwell.PT:= T#100ms;
	Weld_Dwell();

	(*Trigger Capture for Previous LVDT Data*)
	Trig_NutLVDT.CLK:= Weld_Dwell.Q;
	Trig_NutLVDT();
	IF Trig_NutLVDT.Q
		THEN
		IF Option_InScaledValues THEN
			NutPrev_Scaled:= LVDT_Scaled;
		ELSE
			NutPrev_Raw:= Raw_Transducer;
		END_IF;
	END_IF;

	(*Set Nut LVDT Limits Based on Previous LVDT Measurement*)
	IF Save_Nut_Conf THEN
		IF Option_InScaledValues THEN
			(*Scaled Mode*)
			IF (NutPrev_Scaled + 0.5) < 22 THEN
				Nut_UpperLimit[Model_ID]:= NutPrev_Scaled + 0.5;		(*NOTE - JAU - Determined value of 0.5mm by placing M6 nut upside down vs right way up*)
			END_IF;
			IF (NutPrev_Scaled - 0.5) > 0 THEN
				Nut_LowerLimit[Model_ID]:= NutPrev_Scaled -  0.5;
			END_IF;
			(*Unscaled Mode*)
		ELSE	
			Nut_UpperLimit[Model_ID]:= NutPrev_Raw + 300;			(*NOTE - JAU - Determined value of 300 by placing M6 nut upside down vs right way up*)
			Nut_LowerLimit[Model_ID]:= NutPrev_Raw -  300;
		END_IF;
	END_IF;


	(*Creates Prompt and Button Flash on UI IF values between PLC and UI Numeric Inputs do not match*)
	IF (Nut_UpperLimit[Model_ID] = NutInput_UpperLimit[Model_ID] AND (Nut_UpperLimit[Model_ID] <> 0))
	AND (Nut_LowerLimit[Model_ID] = NutInput_LowerLimit[Model_ID] AND (Nut_LowerLimit[Model_ID] <>0))
		THEN
			LVDT_Saved:= TRUE;
	ELSE
			LVDT_Saved:= FALSE;
	END_IF;

	(*Part Present Limit Checks - Allows Weld Schedule to Proceed with Weld - Nut Orientation OK*)
	IF (Model_ID<>0) AND Weld_Dwell.Q THEN
		IF Option_InScaledValues THEN
		NutOK:= (LVDT_Scaled<= Nut_UpperLimit[Model_ID])
					AND (LVDT_Scaled>= Nut_LowerLimit[Model_ID]);
		ELSE		
		NutOK:= (Raw_Transducer<= Nut_UpperLimit[Model_ID])
								AND (Raw_Transducer>= Nut_LowerLimit[Model_ID]);
		END_IF;
	ELSIF Weld_Complete OR Reset_NutOK
		THEN
		NutOK:= FALSE;
	END_IF;





	(*Move Previous LVDT Measurements in Storage Array*)
	Store.CLK:= Weld_Dwell.Q;
	Store();
	IF Store.Q
		THEN
			NutWeld_Store[30]:= NutWeld_Store[29];
			NutWeld_Store[29]:= NutWeld_Store[28];
			NutWeld_Store[28]:= NutWeld_Store[27];
			NutWeld_Store[27]:= NutWeld_Store[26];
			NutWeld_Store[26]:= NutWeld_Store[25];
			NutWeld_Store[25]:= NutWeld_Store[24];
			NutWeld_Store[24]:= NutWeld_Store[23];
			NutWeld_Store[23]:= NutWeld_Store[22];
			NutWeld_Store[22]:= NutWeld_Store[21];
			NutWeld_Store[21]:= NutWeld_Store[20];
			NutWeld_Store[20]:= NutWeld_Store[19];
			NutWeld_Store[19]:= NutWeld_Store[18];
			NutWeld_Store[18]:= NutWeld_Store[17];
			NutWeld_Store[17]:= NutWeld_Store[16];
			NutWeld_Store[16]:= NutWeld_Store[15];
			NutWeld_Store[15]:= NutWeld_Store[14];
			NutWeld_Store[14]:= NutWeld_Store[13];
			NutWeld_Store[13]:= NutWeld_Store[12];
			NutWeld_Store[12]:= NutWeld_Store[11];
			NutWeld_Store[11]:= NutWeld_Store[10];
			NutWeld_Store[10]:= NutWeld_Store[9];
			NutWeld_Store[9]:= NutWeld_Store[8];
			NutWeld_Store[8]:= NutWeld_Store[7];
			NutWeld_Store[7]:= NutWeld_Store[6];
			NutWeld_Store[6]:= NutWeld_Store[5];
			NutWeld_Store[5]:= NutWeld_Store[4];
			NutWeld_Store[4]:= NutWeld_Store[3];
			NutWeld_Store[3]:= NutWeld_Store[2];
			NutWeld_Store[2]:= NutWeld_Store[1];
			NutWeld_Store[1]:= NutPrev_Raw;
	END_IF;

END_FUNCTION_BLOCK

// ---- POUs/FUNs/FUN_GTAC_Scaling.TcPOU
(*General scaling function
	author: Brent Lekx-Toniolo OF Sodecia GTAC
	date: November 2016
	version 1.0
		- initial concept
	Last Edit: 17-Nov-2016, b.lekx-toniolo

*)


FUNCTION FUN_GTAC_Scaling : REAL
VAR_INPUT
	Unscaled_Data: REAL;
	Unscaled_LowerLimit: REAL;
	Unscaled_UpperLimit: REAL;
	Scaled_LowerLimit: REAL;
	Scaled_UpperLimit: REAL;

END_VAR
VAR
	Unscaled_Span: REAL;
	Scaled_Span: REAL;
	Scaling_Factor: REAL;
	Offset: REAL;


END_VAR

(*Calc Span of Scaled Input Values*)
	IF Scaled_UpperLimit > Scaled_LowerLimit
		THEN
		Scaled_Span:= Scaled_UpperLimit - Scaled_LowerLimit;
	END_IF;

(*Calc Span of Unscaled Input Values*)
	IF Unscaled_UpperLimit > Unscaled_LowerLimit
		THEN
		Unscaled_Span:= Unscaled_UpperLimit - Unscaled_LowerLimit;
	END_IF;

(*Calc Scaling Factor between two scales*)
	IF Unscaled_Span>0
		THEN
		Scaling_Factor:= Scaled_Span / Unscaled_Span;
	END_IF;

(*Calc Offset using data above using  y = mx+b with b unknown for offset*)
(*Scaled_LowerLimit = Scaling_Factor  * Unscaled_LowerLimit + b*)
	Offset:= 0 - ((Scaling_Factor * Unscaled_LowerLimit) - Scaled_LowerLimit);

(*Return Scaled Data Based on above spans and offset value*)
	FUN_GTAC_Scaling:= ((Scaling_Factor * Unscaled_Data) + Offset);




	(*Place limits on output to prevent over/underscaling*)
	IF FUN_GTAC_Scaling > Scaled_UpperLimit
		THEN
			FUN_GTAC_Scaling:= Scaled_UpperLimit;
	ELSIF FUN_GTAC_Scaling < Scaled_LowerLimit
		THEN
			FUN_GTAC_Scaling:= Scaled_LowerLimit;
	END_IF;

END_FUNCTION

// ---- POUs/FBs/FB_SIC_MarkProfi_20200727.TcPOU
(*FB for use with a SIC Dot Peen Marking System.

Revision
------------------------------------------------------------------------------
	Version 20161124:
	- Initial concept, R.Remillard
	Version 20170223:
	- Added Enable_Motion, J.Vandongen and R.Remillard
	Version 20200727
	-Rebuilt FB for new ProfibusV2 SIC Version C.Drees

*)

FUNCTION_BLOCK FB_SIC_MarkProfi_20200727

VAR_INPUT
	Enable_Motion:						BOOL;
	Start_bool:							BOOL;
	ResetError_bool:						BOOL;
	LoadFile_bool:						BOOL;
	FileName_string:						STRING(12);		(*Max 4 character File Name for V1, Max 12 Character File Name for V2*)
	CompleteReset_bool:					BOOL;
	Bypass_bool:							BOOL;
	Retry_Enable:						BOOL;
	Comm_Method:						INT;(* 1 - V1(RS232 Mode), 2- V2(Full Profibus Comms)*)
	Variables: 							ARRAY [1..11] OF STRING(16);


END_VAR

VAR

	Txx_Internal_ProfiMaster AT %I*: 		udt_EL6731;

	SICMarker_Inputs AT %I*:				udt_SIC_Profi_Input_20200727;
	SICMarker_Outputs AT %Q*:			udt_SIC_Profi_Output_20200727;

	StringLength:							INT;

	LoadChar:							ARRAY [0..11] OF 	BYTE;
	FileChar:								ARRAY [0..11] OF	STRING(1);
	VarByte:								ARRAY [0..15] OF 	BYTE;
	VarChar:								ARRAY [0..15] OF	STRING(1);


	Retry:								BOOL;
	Retry_TMR:							TON;

	StartRtrig:							R_TRIG;
	LastDotRTrig:							R_TRIG;
	AtHomeRtrig:							R_TRIG;
	X:									INT;
	Y:									INT;
	AllVariablesOK: BOOL;
	LoadFileOK: BOOL;
	
END_VAR

VAR_OUTPUT

	DpState:								INT;
	Profinode_OK_bool:					BOOL;

	SIC_Running_bool:					BOOL;
	LastDot_bool:							BOOL;
	BackHome_bool:						BOOL;
	Complete_bool:						BOOL;

	DataReceived_string:					STRING;

END_VAR

(*Check Prifinode is OK*)
Profinode_OK_bool:= SICMarker_Inputs.Inputs.DpState = 0;
DpState:= SICMarker_Inputs.Inputs.DpState;

CASE Comm_Method OF
1:
(*------------------------------------------------------------------------------------------------------------------------------------------------*)
(*Load required command in SIC unit*)
IF Start_bool AND NOT Bypass_bool AND NOT Retry_TMR.Q
	THEN
		(*run[CR][LF] command to SIC Controller*)
		SICMarker_Outputs.Output1_0[0] := 255;			(*FF Hex*)
		SICMarker_Outputs.Output1_0[1]:= 82;				(*R ASCII*)
		SICMarker_Outputs.Output1_0[2]:= 85;				(*U ASCII*)
		SICMarker_Outputs.Output1_0[3]:= 78;				(*N ACCII*)
		SICMarker_Outputs.Output1_0[4]:= 13;				(*[CR] ASCII*)
		SICMarker_Outputs.Output1_0[5]:= 10;				(*[LF] ASCII*)
		SICMarker_Outputs.Output1_0[6]:= 0;
		SICMarker_Outputs.Output1_0[7]:= 0;
		SICMarker_Outputs.Output1_0[8]:= 0;
		SICMarker_Outputs.Output1_0[9]:= 0;
		SICMarker_Outputs.Output1_0[10]:= 0;
		SICMarker_Outputs.Output1_0[11]:= 0;
		SICMarker_Outputs.Output1_0[12]:= 0;
		SICMarker_Outputs.Output1_0[13]:= 0;
		SICMarker_Outputs.Output1_0[14]:= 0;
		SICMarker_Outputs.Output1_0[15]:= 0;

ELSIF (ResetError_bool OR CompleteReset_bool) AND NOT Start_bool AND NOT SIC_Running_bool
	THEN
		(*reseterror[CR][LF] command to SIC Controller*)
		SICMarker_Outputs.Output1_0[0]:= 255;				(*FF Hex*)
		SICMarker_Outputs.Output1_0[1]:= 82;				(*R ASCII*)
		SICMarker_Outputs.Output1_0[2]:= 69;				(*E ASCII*)
		SICMarker_Outputs.Output1_0[3]:= 83;				(*S ASCII*)
		SICMarker_Outputs.Output1_0[4]:= 69;				(*E ASCII*)
		SICMarker_Outputs.Output1_0[5]:= 84;				(*T ASCII*)
		SICMarker_Outputs.Output1_0[6]:= 69;				(*E ASCII*)
		SICMarker_Outputs.Output1_0[7]:= 82;				(*R ASCII*)
		SICMarker_Outputs.Output1_0[8]:= 82;				(*R ASCII*)
		SICMarker_Outputs.Output1_0[9]:= 79;				(*O ASCII*)
		SICMarker_Outputs.Output1_0[10]:= 82;			(*R ASCII*)
		SICMarker_Outputs.Output1_0[11]:= 13;			(*[CR] ASCII*)
		SICMarker_Outputs.Output1_0[12]:= 10;			(*[LF] ASCII*)
		SICMarker_Outputs.Output1_0[13]:= 0;
		SICMarker_Outputs.Output1_0[14]:= 0;
		SICMarker_Outputs.Output1_0[15]:= 0;

ELSIF LoadFile_bool AND NOT Start_bool
	THEN
		(*loadfile[CR][LF] command to SIC Controller*)
		SICMarker_Outputs.Output1_0[0]:= 255;				(*FF Hex*)
		SICMarker_Outputs.Output1_0[1]:= 76;				(*L ASCII*)
		SICMarker_Outputs.Output1_0[2]:= 79;				(*O ASCII*)
		SICMarker_Outputs.Output1_0[3]:= 65;				(*A ASCII*)
		SICMarker_Outputs.Output1_0[4]:= 68;				(*D ASCII*)
		SICMarker_Outputs.Output1_0[5]:= 70;				(*F ASCII*)
		SICMarker_Outputs.Output1_0[6]:= 73;				(*I ASCII*)
		SICMarker_Outputs.Output1_0[7]:= 76;				(*L ASCII*)
		SICMarker_Outputs.Output1_0[8]:= 69;				(*E ASCII*)
		SICMarker_Outputs.Output1_0[9]:= 32;				(*Space ASCII*)
		SICMarker_Outputs.Output1_0[10]:= LoadChar[1];		(*"Char 1" ASCII*)
		SICMarker_Outputs.Output1_0[11]:= LoadChar[2];		(*"Char 2" ASCII*)
		SICMarker_Outputs.Output1_0[12]:= LoadChar[3];		(*"Char 3" ASCII*)
		SICMarker_Outputs.Output1_0[13]:= LoadChar[4];		(*"Char 4" ASCII*)
		SICMarker_Outputs.Output1_0[14]:= LoadChar[5];		(*"Char 5" ASCII*)
		SICMarker_Outputs.Output1_0[15]:= LoadChar[6];		(*"Char 6" ASCII*)

ELSE
		SICMarker_Outputs.Output1_0[0]:= 0;
		SICMarker_Outputs.Output1_0[1]:= 0;
		SICMarker_Outputs.Output1_0[2]:= 0;
		SICMarker_Outputs.Output1_0[3]:= 0;
		SICMarker_Outputs.Output1_0[4]:= 0;
		SICMarker_Outputs.Output1_0[5]:= 0;
		SICMarker_Outputs.Output1_0[6]:= 0;
		SICMarker_Outputs.Output1_0[7]:= 0;
		SICMarker_Outputs.Output1_0[8]:= 0;
		SICMarker_Outputs.Output1_0[9]:= 0;
		SICMarker_Outputs.Output1_0[10]:= 0;
		SICMarker_Outputs.Output1_0[11]:= 0;
		SICMarker_Outputs.Output1_0[12]:= 0;
		SICMarker_Outputs.Output1_0[13]:= 0;
		SICMarker_Outputs.Output1_0[14]:= 0;
		SICMarker_Outputs.Output1_0[15]:= 0;
END_IF;


(*--------------------------------------------------------------------------------------------------------------------------------------------------*)
(*Reply information from SIC control converted to String*)
DataReceived_string:= FUN_GTAC_ASCIItoSTRING(
					SICMarker_Inputs.Input0_0[1],
					SICMarker_Inputs.Input0_0[2],
					SICMarker_Inputs.Input0_0[3],
					SICMarker_Inputs.Input0_0[4],
					SICMarker_Inputs.Input0_0[5],
					SICMarker_Inputs.Input0_0[6],
					SICMarker_Inputs.Input0_0[7],
					SICMarker_Inputs.Input0_0[8],
					SICMarker_Inputs.Input0_0[9],
					SICMarker_Inputs.Input0_0[10],
					SICMarker_Inputs.Input0_0[11],
					SICMarker_Inputs.Input0_0[12],
					SICMarker_Inputs.Input0_0[13],
					SICMarker_Inputs.Input0_0[14],
					SICMarker_Inputs.Input0_0[15],
					0);

(*Capture Responses to RUN command*)
IF DataReceived_string = 'RUN OK$R$N'
	THEN
		SIC_Running_bool:= TRUE;
END_IF;

IF DataReceived_string = '$04'
	THEN
		LastDot_bool:= TRUE;
END_IF;

IF DataReceived_string = '$05'
	THEN
		BackHome_bool:= TRUE;
END_IF;


(*-------------------------------------------------------------------------------------------------------------------------------------------------*)
(*Retry Handling*)
	(*Enable Retry IF Start with SIC Running bool*)
	IF Enable_Motion AND (Start_bool AND NOT BackHome_bool AND NOT SIC_Running_bool) AND Retry_Enable
		THEN
			Retry:=TRUE;
	ELSIF (SIC_Running_bool OR BackHome_bool OR Complete_bool) OR NOT Retry_Enable
		THEN
			Retry:= FALSE;
	END_IF;
	Retry_TMR.PT:= T#2s;
	Retry_TMR.IN:= Retry;
	Retry_TMR();

(*-------------------------------------------------------------------------------------------------------------------------------------------------*)
(*Complete handling*)
(*Complete*)
IF SIC_Running_bool AND LastDot_bool AND BackHome_bool
	THEN
		Complete_bool:= TRUE;

ELSIF Bypass_bool AND Start_bool
	THEN
		Complete_bool:= TRUE;

END_IF;

(*Reset*)
IF CompleteReset_bool OR NOT Enable_Motion
	THEN
		SIC_Running_bool:= FALSE;
		LastDot_bool:= FALSE;
		BackHome_bool:= FALSE;
		Complete_bool:= FALSE;
		Retry:= FALSE;
END_IF;


(*------------------------------------------------------------------------------------------------------------------------------------------------*)
(*Get Length of string*)
StringLength:= LEN (FileName_string);


(*Separate each character from the File Name*)
IF StringLength = 4
	THEN
(*Shift String based on string length*)
		FileChar[1]:= RIGHT (FileName_string,4);
		FileChar[2]:= RIGHT (FileName_string,3);
		FileChar[3]:= RIGHT (FileName_string,2);
		FileChar[4]:= RIGHT (FileName_string,1);

(*Convert file name to ascii characters*)
		LoadChar[1]:= F_ToASC(FileChar[1]);
		LoadChar[2]:= F_ToASC(FileChar[2]);
		LoadChar[3]:= F_ToASC(FileChar[3]);
		LoadChar[4]:= F_ToASC(FileChar[4]);
		LoadChar[5]:= 13;
		LoadChar[6]:= 10;

ELSIF StringLength =3
	THEN
(*Shift String based on string length*)
		FileChar[1]:= RIGHT (FileName_string,3);
		FileChar[2]:= RIGHT (FileName_string,2);
		FileChar[3]:= RIGHT (FileName_string,1);

(*Convert file name to ascii characters*)
		LoadChar[1]:= F_ToASC(FileChar[1]);
		LoadChar[2]:= F_ToASC(FileChar[2]);
		LoadChar[3]:= F_ToASC(FileChar[3]);
		LoadChar[4]:= 13;
		LoadChar[5]:= 10;
		LoadChar[6]:= 0;

ELSIF StringLength =2
	THEN
(*Shift String based on string length*)
		FileChar[1]:= RIGHT (FileName_string,2);
		FileChar[2]:= RIGHT (FileName_string,1);

(*Convert file name to ascii characters*)
		LoadChar[1]:= F_ToASC(FileChar[1]);
		LoadChar[2]:= F_ToASC(FileChar[2]);
		LoadChar[3]:= 13;
		LoadChar[4]:= 10;
		LoadChar[5]:= 0;
		LoadChar[6]:= 0;

ELSIF StringLength =1
	THEN
(*Shift String based on string length*)
		FileChar[1]:= RIGHT (FileName_string,1);

(*Convert file name to ascii characters*)
		LoadChar[1]:= F_ToASC(FileChar[1]);
		LoadChar[2]:= 13;
		LoadChar[3]:= 10;
		LoadChar[4]:= 0;
		LoadChar[5]:= 0;
		LoadChar[6]:= 0;

ELSE
(*Set all to 0*)
		LoadChar[1]:= 0;
		LoadChar[2]:= 0;
		LoadChar[3]:= 0;
		LoadChar[4]:= 0;
		LoadChar[5]:= 0;

END_IF;

2:

(*------------------------------------------------------------------------------------------------------------------------------------------------*)

(*Start Signal to SIC Marker*)
	IF Start_bool AND NOT Bypass_bool AND NOT Retry_TMR.Q THEN
		SICMarker_Outputs.Output1_1[0].0 := TRUE;
	ELSE
		SICMarker_Outputs.Output1_1[0].0 := FALSE;
	END_IF

(*Reset Signal to SIC Marker*)
	IF (ResetError_bool OR CompleteReset_bool) AND NOT Start_bool AND NOT SIC_Running_bool THEN
		SICMarker_Outputs.Output1_1[0].1 := TRUE;
	ELSE
		SICMarker_Outputs.Output1_1[0].1 := FALSE;
	END_IF

(*Load File Signal to SIC Marker*)
	IF LoadFile_bool AND NOT Start_bool THEN
		SICMarker_Outputs.Output1_1[1].7 := TRUE;
	ELSE
		SICMarker_Outputs.Output1_1[1].7 := FALSE;
	END_IF



(*--------------------------------------------------------------------------------------------------------------------------------------------------*)
(*Capture Responses to RUN command*)
	StartRtrig(CLK:=SICMarker_Inputs.Input0_1[1].0);
	IF StartRtrig.Q
		THEN
			SIC_Running_bool:= TRUE;
	END_IF;

(*Capture Last Dot Marked Signal*)
	LastDotRtrig(CLK:=SICMarker_Inputs.Input0_1[0].4 AND SIC_Running_bool);
	IF LastDotRtrig.Q
	THEN
		LastDot_bool:= TRUE;
	END_IF;

IF SICMarker_inputs.Input0_1[0].7 THEN
	LoadFileOK := TRUE;
END_IF


(*Capture Marker At Home Signal*)
	AtHomeRTrig(CLK:=SICMarker_Inputs.Input0_1[0].5 AND SIC_Running_bool);
	IF AtHomeRTrig.Q
		THEN
			BackHome_bool:= TRUE;
	END_IF;


(*-------------------------------------------------------------------------------------------------------------------------------------------------*)
(*Retry Handling*)
	(*Enable Retry IF Start with SIC Running bool*)
	IF Enable_Motion AND (Start_bool AND NOT BackHome_bool AND NOT SIC_Running_bool) AND Retry_Enable
		THEN
			Retry:=TRUE;
	ELSIF (SIC_Running_bool OR BackHome_bool OR Complete_bool) OR NOT Retry_Enable
		THEN
			Retry:= FALSE;
	END_IF;
	Retry_TMR.PT:= T#2s;
	Retry_TMR.IN:= Retry;
	Retry_TMR();

(*-------------------------------------------------------------------------------------------------------------------------------------------------*)
(*Complete handling*)
(*Complete*)
IF SIC_Running_bool AND LastDot_bool AND BackHome_bool
	THEN
		Complete_bool:= TRUE;

ELSIF Bypass_bool AND Start_bool
	THEN
		Complete_bool:= TRUE;

END_IF;

(*Reset*)
IF CompleteReset_bool OR NOT Enable_Motion
	THEN
		SIC_Running_bool:= FALSE;
		LastDot_bool:= FALSE;
		BackHome_bool:= FALSE;
		Complete_bool:= FALSE;
		Retry:= FALSE;
END_IF;


(*------------------------------------------------------------------------------------------------------------------------------------------------*)
(*--------------------------------------------------------------File Load--------------------------------------------------------------------*)
(*------------------------------------------------------------------------------------------------------------------------------------------------*)
(*Get Length of string*)
StringLength:= LEN (FileName_string);

	FOR x := 0 TO 11 DO
		IF X <= StringLength THEN
			FileChar[x]:= RIGHT (FileName_string,StringLength-x);
		END_IF
	END_FOR


(*Convert file name to ascii characters*)

	FOR X:= 0 TO 11 DO
		IF X<= Stringlength THEN
			LoadChar[X]:= F_ToASC(FileChar[X]);
		END_IF
		IF X >Stringlength THEN
			LoadChar[X] :=0;
		END_IF
	END_FOR

(*Moves Filename to Proper Register*)

	SICMarker_Outputs.Output1_1[8]:=	LoadChar[0];
	SICMarker_Outputs.Output1_1[9]:=	LoadChar[1];
	SICMarker_Outputs.Output1_1[10]:=	LoadChar[2];
	SICMarker_Outputs.Output1_1[11]:=	LoadChar[3];
	SICMarker_Outputs.Output1_1[12]:=	LoadChar[4];
	SICMarker_Outputs.Output1_1[13]:=	LoadChar[5];
	SICMarker_Outputs.Output1_1[14]:=	LoadChar[6];
	SICMarker_Outputs.Output1_1[15]:=	LoadChar[7];
	SICMarker_Outputs.Output1_2[0]:=	LoadChar[8];
	SICMarker_Outputs.Output1_2[1]:=	LoadChar[9];
	SICMarker_Outputs.Output1_2[2]:=	LoadChar[10];
	SICMarker_Outputs.Output1_2[3]:=	LoadChar[11];


(*------------------------------------------------------------------------------------------------------------------------------------------------*)
(*-----------------------------------------------------Variable Transfer-----------------------------------------------------------------*)
(*------------------------------------------------------------------------------------------------------------------------------------------------*)

(*Get Length of string*)


	IF Y > 11 OR Y <1 THEN
		Y:=1;
	END_IF

(*Convert Variables name to ascii characters*)


		StringLength:= LEN (Variables[Y]);

		FOR x := 0 TO 11 DO
			IF X <= StringLength THEN
				VarChar[x]:= RIGHT (Variables[Y],StringLength-x);
			END_IF
		END_FOR

		FOR X:= 0 TO 11 DO
			IF X<= Stringlength THEN
				VarByte[X]:= F_ToASC(VarChar[X]);
			END_IF
			IF X >Stringlength THEN
				VarByte[X] :=0;
			END_IF
		END_FOR

	CASE Y OF

	1: (*Set Variable Register PLC01 *)
	SICMarker_Outputs.Output1_3[0]:=	VarByte[0];
	SICMarker_Outputs.Output1_3[1]:=	VarByte[1];
	SICMarker_Outputs.Output1_3[2]:=	VarByte[2];
	SICMarker_Outputs.Output1_3[3]:=	VarByte[3];
	SICMarker_Outputs.Output1_3[4]:=	VarByte[4];
	SICMarker_Outputs.Output1_3[5]:=	VarByte[5];
	SICMarker_Outputs.Output1_3[6]:=	VarByte[6];
	SICMarker_Outputs.Output1_3[7]:=	VarByte[7];
	SICMarker_Outputs.Output1_3[8]:=	VarByte[8];
	SICMarker_Outputs.Output1_3[9]:=	VarByte[9];
	SICMarker_Outputs.Output1_3[10]:=	VarByte[10];
	SICMarker_Outputs.Output1_3[11]:=	VarByte[11];
	SICMarker_Outputs.Output1_3[12]:=	VarByte[12];
	SICMarker_Outputs.Output1_3[13]:=	VarByte[13];
	SICMarker_Outputs.Output1_3[14]:=	VarByte[14];
	SICMarker_Outputs.Output1_3[15]:=	VarByte[15];
	SICMarker_Outputs.Output1_1[4].0 :=TRUE;

	2:  (*Set Variable Register PLC02 *)
	SICMarker_Outputs.Output1_4[0]:=	VarByte[0];
	SICMarker_Outputs.Output1_4[1]:=	VarByte[1];
	SICMarker_Outputs.Output1_4[2]:=	VarByte[2];
	SICMarker_Outputs.Output1_4[3]:=	VarByte[3];
	SICMarker_Outputs.Output1_4[4]:=	VarByte[4];
	SICMarker_Outputs.Output1_4[5]:=	VarByte[5];
	SICMarker_Outputs.Output1_4[6]:=	VarByte[6];
	SICMarker_Outputs.Output1_4[7]:=	VarByte[7];
	SICMarker_Outputs.Output1_4[8]:=	VarByte[8];
	SICMarker_Outputs.Output1_4[9]:=	VarByte[9];
	SICMarker_Outputs.Output1_4[10]:=	VarByte[10];
	SICMarker_Outputs.Output1_4[11]:=	VarByte[11];
	SICMarker_Outputs.Output1_4[12]:=	VarByte[12];
	SICMarker_Outputs.Output1_4[13]:=	VarByte[13];
	SICMarker_Outputs.Output1_4[14]:=	VarByte[14];
	SICMarker_Outputs.Output1_4[15]:=	VarByte[15];
	SICMarker_Outputs.Output1_1[4].1 :=TRUE;

	3:  (*Set Variable Register PLC03 *)
	SICMarker_Outputs.Output1_5[0]:=	VarByte[1];
	SICMarker_Outputs.Output1_5[1]:=	VarByte[2];
	SICMarker_Outputs.Output1_5[2]:=	VarByte[3];
	SICMarker_Outputs.Output1_5[3]:=	VarByte[4];
	SICMarker_Outputs.Output1_5[4]:=	VarByte[5];
	SICMarker_Outputs.Output1_5[5]:=	VarByte[6];
	SICMarker_Outputs.Output1_5[6]:=	VarByte[7];
	SICMarker_Outputs.Output1_5[7]:=	VarByte[8];
	SICMarker_Outputs.Output1_5[8]:=	VarByte[9];
	SICMarker_Outputs.Output1_5[9]:=	VarByte[10];
	SICMarker_Outputs.Output1_5[10]:=	VarByte[11];
	SICMarker_Outputs.Output1_5[11]:=	VarByte[12];
	SICMarker_Outputs.Output1_5[12]:=	VarByte[13];
	SICMarker_Outputs.Output1_5[13]:=	VarByte[14];
	SICMarker_Outputs.Output1_5[14]:=	VarByte[15];
	SICMarker_Outputs.Output1_5[15]:=	VarByte[15];
	SICMarker_Outputs.Output1_1[4].2 :=TRUE;

	4: (*Set Variable Register PLC04 *)
	SICMarker_Outputs.Output1_6[0]:=	VarByte[1];
	SICMarker_Outputs.Output1_6[1]:=	VarByte[2];
	SICMarker_Outputs.Output1_6[2]:=	VarByte[3];
	SICMarker_Outputs.Output1_6[3]:=	VarByte[4];
	SICMarker_Outputs.Output1_6[4]:=	VarByte[5];
	SICMarker_Outputs.Output1_6[5]:=	VarByte[6];
	SICMarker_Outputs.Output1_6[6]:=	VarByte[7];
	SICMarker_Outputs.Output1_6[7]:=	VarByte[8];
	SICMarker_Outputs.Output1_6[8]:=	VarByte[9];
	SICMarker_Outputs.Output1_6[9]:=	VarByte[10];
	SICMarker_Outputs.Output1_6[10]:=	VarByte[11];
	SICMarker_Outputs.Output1_6[11]:=	VarByte[12];
	SICMarker_Outputs.Output1_6[12]:=	VarByte[13];
	SICMarker_Outputs.Output1_6[13]:=	VarByte[14];
	SICMarker_Outputs.Output1_6[14]:=	VarByte[15];
	SICMarker_Outputs.Output1_6[15]:=	VarByte[15];
	SICMarker_Outputs.Output1_1[4].3 :=TRUE;

	5: (*Set Variable Register PLC05 *)
	SICMarker_Outputs.Output1_7[0]:=	VarByte[1];
	SICMarker_Outputs.Output1_7[1]:=	VarByte[2];
	SICMarker_Outputs.Output1_7[2]:=	VarByte[3];
	SICMarker_Outputs.Output1_7[3]:=	VarByte[4];
	SICMarker_Outputs.Output1_7[4]:=	VarByte[5];
	SICMarker_Outputs.Output1_7[5]:=	VarByte[6];
	SICMarker_Outputs.Output1_7[6]:=	VarByte[7];
	SICMarker_Outputs.Output1_7[7]:=	VarByte[8];
	SICMarker_Outputs.Output1_7[8]:=	VarByte[9];
	SICMarker_Outputs.Output1_7[9]:=	VarByte[10];
	SICMarker_Outputs.Output1_7[10]:=	VarByte[11];
	SICMarker_Outputs.Output1_7[11]:=	VarByte[12];
	SICMarker_Outputs.Output1_7[12]:=	VarByte[13];
	SICMarker_Outputs.Output1_7[13]:=	VarByte[14];
	SICMarker_Outputs.Output1_7[14]:=	VarByte[15];
	SICMarker_Outputs.Output1_7[15]:=	VarByte[15];
	SICMarker_Outputs.Output1_1[4].4 :=TRUE;

	6: (*Set Variable Register PLC06 *)
	SICMarker_Outputs.Output1_8[0]:=	VarByte[1];
	SICMarker_Outputs.Output1_8[1]:=	VarByte[2];
	SICMarker_Outputs.Output1_8[2]:=	VarByte[3];
	SICMarker_Outputs.Output1_8[3]:=	VarByte[4];
	SICMarker_Outputs.Output1_8[4]:=	VarByte[5];
	SICMarker_Outputs.Output1_8[5]:=	VarByte[6];
	SICMarker_Outputs.Output1_8[6]:=	VarByte[7];
	SICMarker_Outputs.Output1_8[7]:=	VarByte[8];
	SICMarker_Outputs.Output1_8[8]:=	VarByte[9];
	SICMarker_Outputs.Output1_8[9]:=	VarByte[10];
	SICMarker_Outputs.Output1_8[10]:=	VarByte[11];
	SICMarker_Outputs.Output1_8[11]:=	VarByte[12];
	SICMarker_Outputs.Output1_8[12]:=	VarByte[13];
	SICMarker_Outputs.Output1_8[13]:=	VarByte[14];
	SICMarker_Outputs.Output1_8[14]:=	VarByte[15];
	SICMarker_Outputs.Output1_8[15]:=	VarByte[15];
	SICMarker_Outputs.Output1_1[4].5 :=TRUE;

	7:  (*Set Variable Register PLC07 *)
	SICMarker_Outputs.Output1_9[0]:=	VarByte[1];
	SICMarker_Outputs.Output1_9[1]:=	VarByte[2];
	SICMarker_Outputs.Output1_9[2]:=	VarByte[3];
	SICMarker_Outputs.Output1_9[3]:=	VarByte[4];
	SICMarker_Outputs.Output1_9[4]:=	VarByte[5];
	SICMarker_Outputs.Output1_9[5]:=	VarByte[6];
	SICMarker_Outputs.Output1_9[6]:=	VarByte[7];
	SICMarker_Outputs.Output1_9[7]:=	VarByte[8];
	SICMarker_Outputs.Output1_9[8]:=	VarByte[9];
	SICMarker_Outputs.Output1_9[9]:=	VarByte[10];
	SICMarker_Outputs.Output1_9[10]:=	VarByte[11];
	SICMarker_Outputs.Output1_9[11]:=	VarByte[12];
	SICMarker_Outputs.Output1_9[12]:=	VarByte[13];
	SICMarker_Outputs.Output1_9[13]:=	VarByte[14];
	SICMarker_Outputs.Output1_9[14]:=	VarByte[15];
	SICMarker_Outputs.Output1_9[15]:=	VarByte[15];
	SICMarker_Outputs.Output1_1[4].6 :=TRUE;

	8: (*Set Variable Register PLC08 *)
	SICMarker_Outputs.Output1_10[0]:=	VarByte[1];
	SICMarker_Outputs.Output1_10[1]:=	VarByte[2];
	SICMarker_Outputs.Output1_10[2]:=	VarByte[3];
	SICMarker_Outputs.Output1_10[3]:=	VarByte[4];
	SICMarker_Outputs.Output1_10[4]:=	VarByte[5];
	SICMarker_Outputs.Output1_10[5]:=	VarByte[6];
	SICMarker_Outputs.Output1_10[6]:=	VarByte[7];
	SICMarker_Outputs.Output1_10[7]:=	VarByte[8];
	SICMarker_Outputs.Output1_10[8]:=	VarByte[9];
	SICMarker_Outputs.Output1_10[9]:=	VarByte[10];
	SICMarker_Outputs.Output1_10[10]:=	VarByte[11];
	SICMarker_Outputs.Output1_10[11]:=	VarByte[12];
	SICMarker_Outputs.Output1_10[12]:=	VarByte[13];
	SICMarker_Outputs.Output1_10[13]:=	VarByte[14];
	SICMarker_Outputs.Output1_10[14]:=	VarByte[15];
	SICMarker_Outputs.Output1_10[15]:=	VarByte[15];
	SICMarker_Outputs.Output1_1[4].7 :=TRUE;

	9: (*Set Variable Register PLC9 *)
	SICMarker_Outputs.Output1_11[0]:=	VarByte[1];
	SICMarker_Outputs.Output1_11[1]:=	VarByte[2];
	SICMarker_Outputs.Output1_11[2]:=	VarByte[3];
	SICMarker_Outputs.Output1_11[3]:=	VarByte[4];
	SICMarker_Outputs.Output1_11[4]:=	VarByte[5];
	SICMarker_Outputs.Output1_11[5]:=	VarByte[6];
	SICMarker_Outputs.Output1_11[6]:=	VarByte[7];
	SICMarker_Outputs.Output1_11[7]:=	VarByte[8];
	SICMarker_Outputs.Output1_11[8]:=	VarByte[9];
	SICMarker_Outputs.Output1_11[9]:=	VarByte[10];
	SICMarker_Outputs.Output1_11[10]:=	VarByte[11];
	SICMarker_Outputs.Output1_11[11]:=	VarByte[12];
	SICMarker_Outputs.Output1_11[12]:=	VarByte[13];
	SICMarker_Outputs.Output1_11[13]:=	VarByte[14];
	SICMarker_Outputs.Output1_11[14]:=	VarByte[15];
	SICMarker_Outputs.Output1_11[15]:=	VarByte[15];
	SICMarker_Outputs.Output1_1[5].0 :=TRUE;

	10: (*Set Variable Register PLC10 *)
	SICMarker_Outputs.Output1_12[0]:=	VarByte[1];
	SICMarker_Outputs.Output1_12[1]:=	VarByte[2];
	SICMarker_Outputs.Output1_12[2]:=	VarByte[3];
	SICMarker_Outputs.Output1_12[3]:=	VarByte[4];
	SICMarker_Outputs.Output1_12[4]:=	VarByte[5];
	SICMarker_Outputs.Output1_12[5]:=	VarByte[6];
	SICMarker_Outputs.Output1_12[6]:=	VarByte[7];
	SICMarker_Outputs.Output1_12[7]:=	VarByte[8];
	SICMarker_Outputs.Output1_12[8]:=	VarByte[9];
	SICMarker_Outputs.Output1_12[9]:=	VarByte[10];
	SICMarker_Outputs.Output1_12[10]:=	VarByte[11];
	SICMarker_Outputs.Output1_12[11]:=	VarByte[12];
	SICMarker_Outputs.Output1_12[12]:=	VarByte[13];
	SICMarker_Outputs.Output1_12[13]:=	VarByte[14];
	SICMarker_Outputs.Output1_12[14]:=	VarByte[15];
	SICMarker_Outputs.Output1_12[15]:=	VarByte[15];

	(*Set Variable in SIC Marker Boolean *)
	SICMarker_Outputs.Output1_1[5].1 :=TRUE;

	END_CASE

	(*Increase Variable counter *)
	IF Y < 10 THEN
		Y:=Y+1;
	END_IF

	(*Wait for all PLC variables to match their registers *)
	IF Y > 10 THEN
		AllVariablesOK := (SICMarker_Inputs.Input0_1[2].0  OR Variables[1] = '')
					AND (SICMarker_Inputs.Input0_1[2].1 OR Variables[2] = '')
					AND (SICMarker_Inputs.Input0_1[2].2 OR Variables[3] = '') 
					AND (SICMarker_Inputs.Input0_1[2].3 OR Variables[4] = '')
					AND (SICMarker_Inputs.Input0_1[2].4 OR Variables[5] = '') 
					AND (SICMarker_Inputs.Input0_1[2].5 OR Variables[6] = '')
					AND (SICMarker_Inputs.Input0_1[2].6 OR Variables[7] = '')
					AND (SICMarker_Inputs.Input0_1[2].7 OR Variables[8] = '')
					AND (SICMarker_Inputs.Input0_1[3].0 OR Variables[9] = '') 
					AND (SICMarker_Inputs.Input0_1[2].1 OR Variables[10] = '');
	END_IF

	(*Reset the Bits to send Variable changes, and Variable Counter *)
	IF Y >= 10 AND LoadFile_bool THEN
		Y:=1;
		SICMarker_Outputs.Output1_1[4] :=0;
		SICMarker_Outputs.Output1_1[5] :=0;
	END_IF

END_CASE

END_FUNCTION_BLOCK

// ---- POUs/FUNs/FUN_GTAC_ASCIItoSTRING.TcPOU
(*Takes up to 16 ASCII codes and packs into a STRING return
	author: Brent Lekx-Toniolo and Rob Remillard Of Sodecia GTAC
	date: Nov 2016
	version 1.0
		- initial concept


	Last Edit: 28-Nov-2016, blt/rr
*)




FUNCTION FUN_GTAC_ASCIItoSTRING : STRING
VAR_INPUT
	ASCII_1: BYTE;
	ASCII_2: BYTE;
	ASCII_3: BYTE;
	ASCII_4: BYTE;
	ASCII_5: BYTE;
	ASCII_6: BYTE;
	ASCII_7: BYTE;
	ASCII_8: BYTE;
	ASCII_9: BYTE;
	ASCII_10: BYTE;
	ASCII_11: BYTE;
	ASCII_12: BYTE;
	ASCII_13: BYTE;
	ASCII_14: BYTE;
	ASCII_15: BYTE;
	ASCII_16: BYTE;

END_VAR
VAR

	Chars: ARRAY [1..16] OF STRING[1];
	StringArray: ARRAY [1..16] OF STRING[16];


END_VAR

(*-------------------------------------------------------------------------- Convert Ascis Codes to Chars ----------------------------------------------*)
Chars[1]:= F_ToCHR( ASCII_1);
Chars[2]:= F_ToCHR( ASCII_2);
Chars[3]:= F_ToCHR( ASCII_3);
Chars[4]:= F_ToCHR( ASCII_4);
Chars[5]:= F_ToCHR( ASCII_5);
Chars[6]:= F_ToCHR( ASCII_6);
Chars[7]:= F_ToCHR( ASCII_7);
Chars[8]:= F_ToCHR( ASCII_8);
Chars[9]:= F_ToCHR( ASCII_9);
Chars[10]:= F_ToCHR( ASCII_10);
Chars[11]:= F_ToCHR( ASCII_11);
Chars[12]:= F_ToCHR( ASCII_12);
Chars[13]:= F_ToCHR( ASCII_13);
Chars[14]:= F_ToCHR( ASCII_14);
Chars[15]:= F_ToCHR( ASCII_15);
Chars[16]:= F_ToCHR( ASCII_16);

(*-------------------------------------------------------------------------- Load Chars to String Return ----------------------------------------------*)

StringArray[16]:= CONCAT(Chars[15],Chars[16]);
StringArray[15]:= CONCAT(Chars[14],StringArray[16]);
StringArray[14]:= CONCAT(Chars[13],StringArray[15]);
StringArray[13]:= CONCAT(Chars[12],StringArray[14]);
StringArray[12]:= CONCAT(Chars[11],StringArray[13]);
StringArray[11]:= CONCAT(Chars[10],StringArray[12]);
StringArray[10]:= CONCAT(Chars[9],StringArray[11]);
StringArray[9]:= CONCAT(Chars[8],StringArray[10]);
StringArray[8]:= CONCAT(Chars[7],StringArray[9]);
StringArray[7]:= CONCAT(Chars[6],StringArray[8]);
StringArray[6]:= CONCAT(Chars[5],StringArray[7]);
StringArray[5]:= CONCAT(Chars[4],StringArray[6]);
StringArray[4]:= CONCAT(Chars[3],StringArray[5]);
StringArray[3]:= CONCAT(Chars[2],StringArray[4]);
StringArray[2]:= CONCAT(Chars[1],StringArray[3]);

(*------------------------------------------------------ Return ----------------------------------------*)

FUN_GTAC_ASCIItoSTRING:= StringArray[2];

END_FUNCTION

// ---- POUs/FBs/FB_Trumpf_20180125.TcPOU
(*FB for use with Trumpf Laser Weld Controller. Programmed to a TruDisk5001 Unit:
	Original Author(s): Justin Vandongen of Sodecia GTAC; 
------------------------------------------------------------------------------------------
REVISION NOTES:
	Version 20171002
		- Initial Concept, j.vandongen
	Verson 20180125
		- added in some additional fault logic as some scenarios are not captured, j.vandongen

------------------------------------------------------------------------------------------
*)



FUNCTION_BLOCK FB_Trumpf_20180125
	VAR_INPUT
		Enable_Motion: BOOL;
		Safety_RST: BOOL;				(*Used to reset TwinSAFE Faults*)
		All_Safeties_OK: BOOL;
		Prev_EcatNode_Present: BOOL;

		(*Word 0*)
		Request_Laser: BOOL; 			(*Word 0.0*)
		Pilot_Laser_On: BOOL;				(*Word 0.1*)
		Unsync_Pstart: BOOL;				(*Word 0.2*)
		Simulation: BOOL;					(*Word 0.3*)
		(*reserved*)						(*Word 0.4*)
		Inquiry1: BOOL;					(*Word 0.5*)
		Inquiry2: BOOL;					(*Word 0.6*)
		Fault_EXT: BOOL;					(*Word 0.7*)
		Reset: BOOL;						(*Word 0.8*)
		Prog_Stop: BOOL; 				(*Word 0.9*)
		Pstart_Dyn: BOOL;					(*Word 0.10*)
		Pstart_Statical: BOOL; 				(*Word 0.11*)
		Laser_Standby: BOOL;				(*Word 0.12*)
		Laser_on: BOOL;					(*Word 0.13*)
		Lock_Operating_Panel: BOOL; 		(*Word 0.14*)
		Ext_Activation: BOOL;				(*Word 0.15*)

		(*Word 1*)
		Program_No:	UINT;				(*Word 1.0 - Word 1.7*)
		Light_Path_No:UINT;				(*Word 1.8 - Word 1.15*)

		(*Word 2*)
		Laser_No: UINT;					(*Word 2.0 - Word 2.7*)
		AD_No: UINT;					(*Word 2.8 - Word 2.15*)

		(*Word 3 - 63*)
		(*Parameters for laser, PFO and cutting. This will be handled inside TruControl*)


	END_VAR

	VAR
	(*Hardware Data Types*)
		LSRT01 AT %I*: udt_EL6692_20121204;	(*EtherCAT bridge for Laser controller*)
	(*Develope EtherCAT Interface*)
		In_From_ECAT AT %I*: udt_EtherCat_Trumpf_InputWords_20171002;
		Out_To_ECAT AT %Q*: udt_EtherCat_Trumpf_OutputWords_20171002;

	(* Nodes/Interface States*)
		DiscreteNode_OK: BOOL;
		EtherCATNode_OK: BOOL;
		EtherCATConn_OK: BOOL;

	(*Cable Break Warning Flags*)
		ECatSlave_Cable_Breaks: UDINT;
		EL6692_NotPresent :BOOL;			(*Bridge Terminal is not on Bus when expected*)
		EL6692_PortC_MissingLink: BOOL;


	(*Delay Timers*)
		Delay_Time0: TON;
		Delay_Time1: TON;
		Delay_Time2: TON;
		Delay_Time3: TON;
		Delay_Time4: TON;

	(*Internal Variables*)
		Laser_Power_Prev: UDINT;
		Energy_Prev: UDINT;
		Laser_Power_CurrentVal: UDINT;
		Energy_CurrentVal: UDINT;

	(*Fault Timers and flags*)
		Ext_Act_Fault_TMR: TON;
		Laser_On_Fault_TMR: TON;
		Req_Laser_Fault_TMR: TON;

	END_VAR

	VAR_OUTPUT
		FB_OK: BOOL;

		Input_Image:udt_EtherCat_Trumpf_InputWords_20171002;
		Output_Image:udt_EtherCat_Trumpf_OutputWords_20171002;

		Discrete_Image: udt_TrumpfImage_20171017;

		Laser_Faulted: BOOL;
		Welding_Complete: BOOL;

		(*Word 0*)
		Laser_Warning_Lamp_Is_On: BOOL;		(*Word 0.0*)
		Pilot_Laser_Is_On: BOOL;				(*Word 0.1*)
		Power_Limit: BOOL; 					(*Word 0.2*)
		Laser_Assigned: BOOL; 				(*Word 0.3*)
		Fault_Laser: BOOL;					(*Word 0.4*)
		Monitoring: BOOL; 						(*Word 0.5*)
		Sik_Open: BOOL;						(*Word 0.6*)
		Set_3: BOOL;							(*Word 0.7*)
		Set_2: BOOL;							(*Word 0.8*)
		Set_1:BOOL;							(*Word 0.9*)
		Prog_Cancelled: BOOL;				(*Word 0.10*)
		Prog_Completed: BOOL;				(*Word 0.11*)
		Prog_Active: BOOL;					(*Word 0.12*)
		Laser_Ready: BOOL;					(*Word 0.13*)
		Laser_Is_On: BOOL;					(*Word 0.14*)
		Ext_Activation_Active: BOOL;			(*Word 0.15*)

		(*Word 1*)
		Program_No_ACK: UINT;				(*Word 1.0 - 1.7*)
		Light_Path_No_ACK: UINT;				(*Word 1.8 - 1.15*)

		(*Word 2*)
		Shutter_Switch: UINT;					(*Word 2.0 - 2.7*)
		Fault_Slot: BOOL;						(*Word 2.8*)
		Monitoring_Slot: BOOL;					(*Word 2.9*)
		(*reserved*)							(*Word 2.10*)
		Focusing_Optics_Avail: BOOL;			(*Word 2.11*)
		Focusing_Optics_Ready: BOOL;			(*Word 2.12*)
		Application_Values_In_Range: BOOL;	(*Word 2.13*)
		Protective_Glass_Soiled: BOOL;			(*Word 2.14*)
		Protective_Glass_Life_Reached: BOOL;	(*Word 2.15*)

		(*Word 3*)
		Measuring_Value_Out_Active: BOOL;		(*Word 3.0*)
		Maintenance: BOOL;					(*Word 3.1*)
		Chiller_Rinsing_Heating: BOOL;			(*Word 3.2*)
		Calibration_Self_Test: BOOL;			(*Word 3.3*)
		Alive_Tick: BOOL;						(*Word 3.4*)
		Ext_Cooling_On: BOOL;				(*Word 3.5*)
		(*reserved*)							(*Word 3.6*)
		(*reserved*)							(*Word 3.7*)
		Laser_No_ACK: UINT;					(*Word 3.8 - 3.15*)

		(*Word 4*)
		Message_Num: UINT;					(*Word 4.0 - 4.7*)
		Message_ID: UINT;					(*Word 4.8 - 4.15*)

		(*Word 5*)
		Measuring_Value_ID: UINT;				(*Word 5*)

		(*Word 6*)
		Laser_Power: UINT;					(*Word 6*)

		(*Word 7*)
		Energy: UINT;						(*Word 7*)

		(*Word 8 - 63*)
		(*Other parameters not currently being used*)



	END_VAR

	(*Set FB_OK to True*)
	FB_OK:= TRUE;

(*$$$$$$$$$$$$$$$$$$$$$$$$$$$$$$$$$$$$$$$$$$$$$$$$Gather Status Of Hardware $$$$$$$$$$$$$$$$$$$$$$$$$$$$$$$$$$$$$$$$$$$$$$$$$$$$*)

	IF LSRT01.InfoData.State=8
		THEN DiscreteNode_OK:= TRUE;
	ELSE DiscreteNode_OK:= FALSE;
	END_IF;

	(*Develop Port Connection Warning Flags*)
	IF LSRT01.InfoData.State=257 (*State Machine for Slave Not Present*)
		THEN EL6692_NotPresent:= TRUE;
	ELSE EL6692_NotPresent := FALSE;
	END_IF;

	IF LSRT01.InfoData.State= 9224 (*State Machine for Link Missing at Port C*)
		THEN EL6692_PortC_MissingLink:= TRUE; (*PortC is OUT Port*)
	ELSE EL6692_PortC_MissingLink := FALSE;
	END_IF;

	(*Wrap up break Flags to Variable for shipment to UI*)
	ECatSlave_Cable_Breaks.0:= EL6692_NotPresent AND Prev_EcatNode_Present;
	ECatSlave_Cable_Breaks.1:= EL6692_PortC_MissingLink;


(*$$$$$$$$$$$$$$$$$$$$$$$$$$$$$$$$$$$$$$$$$$$$$$$$$$$$Gather All Standard and System Inputs $$$$$$$$$$$$$$$$$$$$$$$$$$$$$$$$$$$$$$$$$$$$$$$$$$$$$$$$$$$$$*)
(* ------------------------- System Inputs Section ----------------------*)

	(*In From EtherCAT Word 0*)
		Laser_Warning_Lamp_Is_On:= In_From_ECAT.Laser_Out[0].0;
		Pilot_Laser_Is_On:= In_From_ECAT.Laser_Out[0].1;
		Power_Limit:= In_From_ECAT.Laser_Out[0].2;
		Laser_Assigned:= In_From_ECAT.Laser_Out[0].3;
		Fault_Laser:= In_From_ECAT.Laser_Out[0].4;
		Monitoring:= In_From_ECAT.Laser_Out[0].5;
		Sik_Open:= In_From_ECAT.Laser_Out[0].6;
		Set_3:= In_From_ECAT.Laser_Out[0].7;
		Set_2:= In_From_ECAT.Laser_Out[0].8;
		Set_1:= In_From_ECAT.Laser_Out[0].9;
		Prog_Cancelled:= In_From_ECAT.Laser_Out[0].10;
		Prog_Completed:= In_From_ECAT.Laser_Out[0].11;
		Prog_Active:= In_From_ECAT.Laser_Out[0].12;
		Laser_Ready:= In_From_ECAT.Laser_Out[0].13;
		Laser_Is_On:= In_From_ECAT.Laser_Out[0].14;
		Ext_Activation_Active:= In_From_ECAT.Laser_Out[0].15;

	(*In From EtherCAT Word 1*)
		Program_No_ACK.0:= In_From_ECAT.Laser_Out[1].0;
		Program_No_ACK.1:= In_From_ECAT.Laser_Out[1].1;
		Program_No_ACK.2:= In_From_ECAT.Laser_Out[1].2;
		Program_No_ACK.3:= In_From_ECAT.Laser_Out[1].3;
		Program_No_ACK.4:= In_From_ECAT.Laser_Out[1].4;
		Program_No_ACK.5:= In_From_ECAT.Laser_Out[1].5;
		Program_No_ACK.6:= In_From_ECAT.Laser_Out[1].6;
		Program_No_ACK.7:= In_From_ECAT.Laser_Out[1].7;
		Light_Path_No_ACK.0:= In_From_ECAT.Laser_Out[1].8;
		Light_Path_No_ACK.1:= In_From_ECAT.Laser_Out[1].9;
		Light_Path_No_ACK.2:= In_From_ECAT.Laser_Out[1].10;
		Light_Path_No_ACK.3:= In_From_ECAT.Laser_Out[1].11;
		Light_Path_No_ACK.4:= In_From_ECAT.Laser_Out[1].12;
		Light_Path_No_ACK.5:= In_From_ECAT.Laser_Out[1].13;
		Light_Path_No_ACK.6:= In_From_ECAT.Laser_Out[1].14;
		Light_Path_No_ACK.7:= In_From_ECAT.Laser_Out[1].15;

	(*In From EtherCAT Word 2*)
		Shutter_Switch.0:= In_From_ECAT.Laser_Out[2].0;
		Shutter_Switch.1:= In_From_ECAT.Laser_Out[2].1;
		Shutter_Switch.2:= In_From_ECAT.Laser_Out[2].2;
		Shutter_Switch.3:= In_From_ECAT.Laser_Out[2].3;
		Shutter_Switch.4:= In_From_ECAT.Laser_Out[2].4;
		Shutter_Switch.5:= In_From_ECAT.Laser_Out[2].5;
		Shutter_Switch.6:= In_From_ECAT.Laser_Out[2].6;
		Shutter_Switch.7:= In_From_ECAT.Laser_Out[2].7;
		Fault_Slot:= In_From_ECAT.Laser_Out[2].8;
		Monitoring_Slot:= In_From_ECAT.Laser_Out[2].9;
		(*Reserved, not used := In_From_ECAT.Laser_Out[2].10;*)
		Focusing_Optics_Avail:= In_From_ECAT.Laser_Out[2].11;
		Focusing_Optics_Ready:= In_From_ECAT.Laser_Out[2].12;
		Application_Values_In_Range:= In_From_ECAT.Laser_Out[2].13;
		Protective_Glass_Soiled:= In_From_ECAT.Laser_Out[2].14;
		Protective_Glass_Life_Reached:= In_From_ECAT.Laser_Out[2].15;

	(*In From EtherCAT Word 3*)
		Measuring_Value_Out_Active:= In_From_ECAT.Laser_Out[3].0;
		Maintenance:= In_From_ECAT.Laser_Out[3].1;
		Chiller_Rinsing_Heating:= In_From_ECAT.Laser_Out[3].2;
		Calibration_Self_Test:= In_From_ECAT.Laser_Out[3].3;
		Alive_Tick:= In_From_ECAT.Laser_Out[3].4;
		Ext_Cooling_On:= In_From_ECAT.Laser_Out[3].5;
		(*Reserved, not used := In_From_ECAT.Laser_Out[3].6;*)
		(*Reserved, not used := In_From_ECAT.Laser_Out[3].7;*)
		Laser_No_ACK.0:= In_From_ECAT.Laser_Out[3].8;
		Laser_No_ACK.1:= In_From_ECAT.Laser_Out[3].9;
		Laser_No_ACK.2:= In_From_ECAT.Laser_Out[3].10;
		Laser_No_ACK.3:= In_From_ECAT.Laser_Out[3].11;
		Laser_No_ACK.4:= In_From_ECAT.Laser_Out[3].12;
		Laser_No_ACK.5:= In_From_ECAT.Laser_Out[3].13;
		Laser_No_ACK.6:= In_From_ECAT.Laser_Out[3].14;
		Laser_No_ACK.7:= In_From_ECAT.Laser_Out[3].15;

	(*In From EtherCAT Word 4*)
		Message_Num.0:= In_From_ECAT.Laser_Out[4].0;
		Message_Num.1:= In_From_ECAT.Laser_Out[4].1;
		Message_Num.2:= In_From_ECAT.Laser_Out[4].2;
		Message_Num.3:= In_From_ECAT.Laser_Out[4].3;
		Message_Num.4:= In_From_ECAT.Laser_Out[4].4;
		Message_Num.5:= In_From_ECAT.Laser_Out[4].5;
		Message_Num.6:= In_From_ECAT.Laser_Out[4].6;
		Message_Num.7:= In_From_ECAT.Laser_Out[4].7;
		Message_ID.0:= In_From_ECAT.Laser_Out[4].8;
		Message_ID.1:= In_From_ECAT.Laser_Out[4].9;
		Message_ID.2:= In_From_ECAT.Laser_Out[4].10;
		Message_ID.3:= In_From_ECAT.Laser_Out[4].11;
		Message_ID.4:= In_From_ECAT.Laser_Out[4].12;
		Message_ID.5:= In_From_ECAT.Laser_Out[4].13;
		Message_ID.6:= In_From_ECAT.Laser_Out[4].14;
		Message_ID.7:= In_From_ECAT.Laser_Out[4].15;

	(*In From EtherCAT Word 5*)
		Measuring_Value_ID.0:= In_From_ECAT.Laser_Out[5].0;
		Measuring_Value_ID.1:= In_From_ECAT.Laser_Out[5].1;
		Measuring_Value_ID.2:= In_From_ECAT.Laser_Out[5].2;
		Measuring_Value_ID.3:= In_From_ECAT.Laser_Out[5].3;
		Measuring_Value_ID.4:= In_From_ECAT.Laser_Out[5].4;
		Measuring_Value_ID.5:= In_From_ECAT.Laser_Out[5].5;
		Measuring_Value_ID.6:= In_From_ECAT.Laser_Out[5].6;
		Measuring_Value_ID.7:= In_From_ECAT.Laser_Out[5].7;
		Measuring_Value_ID.8:= In_From_ECAT.Laser_Out[5].8;
		Measuring_Value_ID.9:= In_From_ECAT.Laser_Out[5].9;
		Measuring_Value_ID.10:= In_From_ECAT.Laser_Out[5].10;
		Measuring_Value_ID.11:= In_From_ECAT.Laser_Out[5].11;
		Measuring_Value_ID.12:= In_From_ECAT.Laser_Out[5].12;
		Measuring_Value_ID.13:= In_From_ECAT.Laser_Out[5].13;
		Measuring_Value_ID.14:= In_From_ECAT.Laser_Out[5].14;
		Measuring_Value_ID.15:= In_From_ECAT.Laser_Out[5].15;

	(*In From EtherCAT Word 6*)
		Laser_Power.0:= In_From_ECAT.Laser_Out[6].0;
		Laser_Power.1:= In_From_ECAT.Laser_Out[6].1;
		Laser_Power.2:= In_From_ECAT.Laser_Out[6].2;
		Laser_Power.3:= In_From_ECAT.Laser_Out[6].3;
		Laser_Power.4:= In_From_ECAT.Laser_Out[6].4;
		Laser_Power.5:= In_From_ECAT.Laser_Out[6].5;
		Laser_Power.6:= In_From_ECAT.Laser_Out[6].6;
		Laser_Power.7:= In_From_ECAT.Laser_Out[6].7;
		Laser_Power.8:= In_From_ECAT.Laser_Out[6].8;
		Laser_Power.9:= In_From_ECAT.Laser_Out[6].9;
		Laser_Power.10:= In_From_ECAT.Laser_Out[6].10;
		Laser_Power.11:= In_From_ECAT.Laser_Out[6].11;
		Laser_Power.12:= In_From_ECAT.Laser_Out[6].12;
		Laser_Power.13:= In_From_ECAT.Laser_Out[6].13;
		Laser_Power.14:= In_From_ECAT.Laser_Out[6].14;
		Laser_Power.15:= In_From_ECAT.Laser_Out[6].15;

	(*In From EtherCAT Word 7*)
		Energy.0:= In_From_ECAT.Laser_Out[7].0;
		Energy.1:= In_From_ECAT.Laser_Out[7].1;
		Energy.2:= In_From_ECAT.Laser_Out[7].2;
		Energy.3:= In_From_ECAT.Laser_Out[7].3;
		Energy.4:= In_From_ECAT.Laser_Out[7].4;
		Energy.5:= In_From_ECAT.Laser_Out[7].5;
		Energy.6:= In_From_ECAT.Laser_Out[7].6;
		Energy.7:= In_From_ECAT.Laser_Out[7].7;
		Energy.8:= In_From_ECAT.Laser_Out[7].8;
		Energy.9:= In_From_ECAT.Laser_Out[7].9;
		Energy.10:= In_From_ECAT.Laser_Out[7].10;
		Energy.11:= In_From_ECAT.Laser_Out[7].11;
		Energy.12:= In_From_ECAT.Laser_Out[7].12;
		Energy.13:= In_From_ECAT.Laser_Out[7].13;
		Energy.14:= In_From_ECAT.Laser_Out[7].14;
		Energy.15:= In_From_ECAT.Laser_Out[7].15;

	(*In From EtherCAT Word  8 - 63*)
		(*Other parameters not currently being used*)






(*$$$$$$$$$$$$$$$$$$$$$$$$$$$$$$$$$$$$$$$$$$$$$$$$$$ Internal Code $$$$$$$$$$$$$$$$$$$$$$$$$$$$$$$$$$$$$$$$$$$$$$$$$$$$$$$$*)


	(*Weld Complete*)
		IF Enable_Motion AND All_Safeties_OK AND Laser_Assigned
			AND (Unsync_Pstart OR Pstart_Dyn OR Pstart_Statical)
			AND Prog_Completed
				THEN Welding_Complete:= TRUE;
		ELSIF NOT Unsync_Pstart AND NOT Pstart_Dyn AND NOT Pstart_Statical
				THEN Welding_Complete:= FALSE;
		END_IF;


	(*Delay Timers for Synchonizing outputs to the laser controller*)
	Delay_Time1(
			IN:= Enable_Motion AND All_Safeties_OK AND Ext_Activation_Active,
			PT:= T#125ms,
			Q=> ,
			ET=> );

	Delay_Time2(
			IN:= Enable_Motion AND All_Safeties_OK AND Laser_Is_On,
			PT:= T#125ms,
			Q=> ,
			ET=> );


	(*Capture Power and Energy results from laser*)
	IF (Unsync_Pstart OR Pstart_Dyn OR Pstart_Statical) AND NOT Prog_Completed
		THEN
		Laser_Power_CurrentVal:= Laser_Power;
		Energy_CurrentVal:= Energy;
	END_IF;

	IF Prog_Completed
		THEN
		Laser_Power_Prev:= Laser_Power_CurrentVal;
		Energy_Prev:= Energy_CurrentVal;
	END_IF;

	Request_Laser:= Enable_Motion AND All_Safeties_OK AND Laser_Is_On AND Delay_Time2.Q;
	Laser_on:= Enable_Motion AND All_Safeties_OK AND Ext_Activation_Active AND Delay_Time1.Q;
 	Ext_Activation:= Enable_Motion AND All_Safeties_OK AND NOT Laser_Faulted;



(*$$$$$$$$$$$$$$$$$$$$$$$$$$$$$$$$$$$$$$$$$$$$$$ Transfer Standard Outputs $$$$$$$$$$$$$$$$$$$$$$$$$$$$$$$$$$$$$$$$$$$*)

	(*Transfer I/O Images for Display On HMI*)
	Input_Image:= In_From_ECAT;
	Output_Image:= Out_To_ECAT;

	Discrete_Image.LSRT01:= LSRT01;
	Discrete_Image.Program_REQ:= Program_No;
	Discrete_Image.Program_ACK:=Program_No_ACK;
	Discrete_Image.Light_Path_REQ:= Light_Path_No;
	Discrete_Image.Light_Path_ACK:= Light_Path_No_ACK;
	Discrete_Image.Laser_No_REQ:= Laser_No;
	Discrete_Image.Laser_No_ACK:= Laser_No_ACK;
	Discrete_Image.Laser_Power:= Laser_Power;
	Discrete_Image.Laser_Power_Prev:= Laser_Power_Prev;
	Discrete_Image.Energy:= Energy;
	Discrete_Image.Energy_Prev:= Energy_Prev;
	Discrete_Image.Faulted:= Laser_Faulted;
	Discrete_Image.Weld_Complete:= Welding_Complete;





	(*--------------- System Outputs to Laser System Inputs -------------------------*)

	(*Out To EtherCAT Word 0*)
		Out_To_ECAT.Laser_In[0].0:= Request_Laser;
		Out_To_ECAT.Laser_In[0].1:= Pilot_Laser_On;
		Out_To_ECAT.Laser_In[0].2:= Unsync_Pstart AND Enable_Motion AND All_Safeties_OK AND Laser_Assigned;
		Out_To_ECAT.Laser_In[0].3:= Simulation;
		(*Out_To_ECAT.Laser_In[0].4:= Reserved;*)
		Out_To_ECAT.Laser_In[0].5:= Inquiry2;
		Out_To_ECAT.Laser_In[0].6:= Inquiry1;
		Out_To_ECAT.Laser_In[0].7:= Fault_EXT;
		Out_To_ECAT.Laser_In[0].8:= Reset AND Laser_Faulted;
		Out_To_ECAT.Laser_In[0].9:= Prog_Stop;
		Out_To_ECAT.Laser_In[0].10:= Pstart_Dyn AND Enable_Motion AND All_Safeties_OK AND Laser_Assigned;
		Out_To_ECAT.Laser_In[0].11:= Pstart_Statical AND Enable_Motion AND All_Safeties_OK AND Laser_Assigned;
		Out_To_ECAT.Laser_In[0].12:= Laser_Standby;
		Out_To_ECAT.Laser_In[0].13:= Laser_on;
		Out_To_ECAT.Laser_In[0].14:= Lock_Operating_Panel;
		Out_To_ECAT.Laser_In[0].15:= Ext_Activation;

	(*Out To EtherCAT Word 1*)
		Out_To_ECAT.Laser_In[1].0:= Program_No.0;
		Out_To_ECAT.Laser_In[1].1:= Program_No.1;
		Out_To_ECAT.Laser_In[1].2:= Program_No.2;
		Out_To_ECAT.Laser_In[1].3:= Program_No.3;
		Out_To_ECAT.Laser_In[1].4:= Program_No.4;
		Out_To_ECAT.Laser_In[1].5:= Program_No.5;
		Out_To_ECAT.Laser_In[1].6:= Program_No.6;
		Out_To_ECAT.Laser_In[1].7:= Program_No.7;
		Out_To_ECAT.Laser_In[1].8:= Light_Path_No.0;
		Out_To_ECAT.Laser_In[1].9:= Light_Path_No.1;
		Out_To_ECAT.Laser_In[1].10:= Light_Path_No.2;
		Out_To_ECAT.Laser_In[1].11:= Light_Path_No.3;
		Out_To_ECAT.Laser_In[1].12:= Light_Path_No.4;
		Out_To_ECAT.Laser_In[1].13:= Light_Path_No.5;
		Out_To_ECAT.Laser_In[1].14:= Light_Path_No.6;
		Out_To_ECAT.Laser_In[1].15:= Light_Path_No.7;

	(*Out To EtherCAT Word 2*)
		Out_To_ECAT.Laser_In[2].0:= Laser_No.0;
		Out_To_ECAT.Laser_In[2].1:= Laser_No.1;
		Out_To_ECAT.Laser_In[2].2:= Laser_No.2;
		Out_To_ECAT.Laser_In[2].3:= Laser_No.3;
		Out_To_ECAT.Laser_In[2].4:= Laser_No.4;
		Out_To_ECAT.Laser_In[2].5:= Laser_No.5;
		Out_To_ECAT.Laser_In[2].6:= Laser_No.6;
		Out_To_ECAT.Laser_In[2].7:= Laser_No.7;
		Out_To_ECAT.Laser_In[2].8:= AD_No.0;
		Out_To_ECAT.Laser_In[2].9:= AD_No.1;
		Out_To_ECAT.Laser_In[2].10:= AD_No.2;
		Out_To_ECAT.Laser_In[2].11:= AD_No.3;
		Out_To_ECAT.Laser_In[2].12:= AD_No.4;
		Out_To_ECAT.Laser_In[2].13:= AD_No.5;
		Out_To_ECAT.Laser_In[2].14:= AD_No.6;
		Out_To_ECAT.Laser_In[2].15:= AD_No.7;

	(*Out To EtherCAT Word 3 - 63*)
		(*Parameters for laser, PFO and cutting. This will be handled inside TruControl*)





	(*Faults*)
		(*External Activation Fault Timer*)
		Ext_Act_Fault_TMR(
					IN:= Ext_Activation AND NOT Ext_Activation_Active,
					PT:= T#5s,
					Q=> ,
					ET=> );

		(*Laser On Fault Timer*)
		Laser_On_Fault_TMR(
					IN:= Laser_on AND NOT Laser_Is_On,
					PT:= T#5s,
					Q=> ,
					ET=> );

		(*Request Laser Fault Timer*)
		Req_Laser_Fault_TMR(
					IN:= Request_Laser AND NOT Laser_Assigned,
					PT:= T#5s,
					Q=> ,
					ET=> );

		(*Gather all Faults*)
		Laser_Faulted:= Fault_Laser
					OR Fault_Slot
					OR Monitoring_Slot
					OR Protective_Glass_Soiled
					OR Prog_Cancelled
					OR Protective_Glass_Life_Reached
					OR Ext_Act_Fault_TMR.Q
					OR Laser_On_Fault_TMR.Q
					OR Req_Laser_Fault_TMR.Q;







(*end*)

END_FUNCTION_BLOCK

// ---- POUs/FBs/FB_GTAC_RollDoor_20190108.TcPOU
(*FB for use with Rite Hite Roll Up Doors

	Original Author(s): Justin Vandongen of Sodecia GTAC.; 
------------------------------------------------------------------------------------------
REVISION NOTES:
	Version 20181023
		- intial concept, J.Vandongen
	Version 20190108
		- modified controls for door close using In_auto and in_manual, j.vandongen
------------------------------------------------------------------------------------------
*)


FUNCTION_BLOCK FB_GTAC_RollDoor_20190108
VAR_INPUT
		Enable_FB: BOOL;
		Enable_Motion: BOOL;
		Enable_Latch: BOOL;

		DoorClose_REQ: BOOL;		(*Request to close the door*)
		DoorOpen_REQ: BOOL;		(*Request to open the door*)

		DoorClosed_Switches: BOOL;	(*Switches to detect Door Closed*)
		DoorOpened_Switches: BOOL;	(*Switches to detect Door opened*)

		Fault_Time: TIME;
END_VAR

VAR
		Door_CloseSR: SR;	(*Latch to Close the door*)
		Door_OpenSR: SR;	(*Latch to Open the door*)

		DoorOpened_TMR: TON;		(*Timer to say door is open, no door open switches*)
		DoorClosed_TMR: TON;	(*Timer to say door is closed*)

		Fault_TMR: TON;

END_VAR

VAR_OUTPUT
		FB_OK: BOOL;

		DoorClose_CMD: BOOL;	(*Command the door to close*)
		DoorOpen_CMD: BOOL;	(*Command the door to open*)
		Door_Closed: BOOL;		(*Door is closed*)
		Door_Opened: BOOL;		(*Door is open*)

		Faulted: BOOL;

END_VAR

	(*Set FB_OK to True*)
	FB_OK:= TRUE;


	(*Set Door to Close*)
	Door_CloseSR(
			SET1:= Enable_Motion AND Enable_Latch AND DoorClose_REQ AND NOT DoorOpen_REQ,
			RESET:= NOT Enable_Motion OR NOT Enable_Latch OR DoorOpen_REQ OR Door_Closed,
			Q1=>
			);

	(*Set Door to Open*)
	Door_OpenSR(
			SET1:= Enable_Latch AND DoorOpen_REQ AND NOT DoorClose_REQ,
			RESET:= NOT Enable_Latch OR DoorClose_REQ OR Door_Opened,
			Q1=>
			);

	(*Output to Open or Close the Door*)
	DoorClose_CMD:= Enable_Motion AND ((Enable_Latch AND Door_CloseSR.Q1) OR (NOT Enable_Latch AND DoorClose_REQ)) AND NOT Door_OpenSR.Q1;
	DoorOpen_CMD:= ((Enable_Latch AND Door_OpenSR.Q1) OR (NOT Enable_Latch AND DoorOpen_REQ)) AND NOT Door_CloseSR.Q1;

	(*Door Opened Timer*)
	DoorOpened_TMR(
			IN:= NOT DoorClosed_Switches AND DoorOpen_CMD,
			PT:= T#2.75s,
			Q=> ,
			ET=>
			);

	(*Door Closed Timer*)
	DoorClosed_TMR(
			IN:= DoorClosed_Switches,
			PT:= T#500ms,
			Q=> ,
			ET=>
			);


	(*Capture Door Closed*)
	IF DoorClosed_Switches AND DoorClosed_TMR.Q
		THEN
			Door_Closed:= TRUE;
			Door_Opened:= FALSE;
	ELSIF NOT DoorClosed_Switches AND DoorOpened_TMR.Q
		THEN
			Door_Closed:= FALSE;
			Door_Opened:= TRUE;
	END_IF;


	(*Capture Door Faults*)
	Fault_TMR(
			IN:= (DoorClose_CMD AND NOT Door_Closed) OR (DoorOpen_CMD AND NOT Door_Opened),
			PT:= Fault_Time,
			Q=> Faulted,
			ET=> );















(*end*)

END_FUNCTION_BLOCK

// ---- POUs/FBs/FB_GTAC_MDxx_20251008.TcPOU
(*FB for use with Rite Hite Roll Up Doors
	Original Author(s): Alan Lopez of Sodecia GTAC.; 
------------------------------------------------------------------------------------------
REVISION NOTES:
	Version 20230718
		- Intial concept, A.Lopez
	Version 20250417
		- Revamped, changed IO for EP rahter then the EL's, r.jones
		- cable break added EP2624
	Version 20251008
		- Revamp per Hardware design requests, b.lekx-toniolo
	Version 20260319
		- Moved DoorClosed_Safety_Switches To Inputs Mapped from Safetys to Std for safety switches, TLK
	

------------------------------------------------------------------------------------------
*)


FUNCTION_BLOCK FB_GTAC_MDxx_20251008
	VAR_INPUT

			(*Internal Input Variables*)
			Enable_Motion: BOOL;
			Safety_RST: BOOL;
			OPxx_RST: BOOL;
			Ecat_Master_AmsNetID: STRING;
			CoE_Read_Trigger: BOOL;
			Enable_Latch: BOOL;
			Prev_EcatNode_Present: BOOL;
			DoorClose_REQ: BOOL;					(*Request to close the door*)
			DoorOpen_REQ: BOOL;						(*Request to open the door*)
			Fault_Time: TIME;
			DoorStop_REQ: BOOL;
			DoorStopped: BOOL;
			DoorClosed_Safety_Switches: BOOL;		(*TLK MOVE TO INPUTS*)
		
	END_VAR

	VAR
		(*Hardware Data Types*)
			(*Develop Discrete Nodes*)
			N01_STAT AT %I*: udt_EP1918_STAT_20250213;		(*EP Based Twinsafe*)
			N01_CMD AT %Q*: udt_EP1918_CMD_20250213;		(*EP Based Twinsafe*)
			N02 AT %I*: udt_EP1008_002_v2;					(*EP Inputs*)
			N03 AT %Q*: udt_EP2624;							(*EP 4ch Relay Output*)
			N03_STAT AT %I*: udt_EP2624_STAT;				(*EP 4ch Relay Output Card Status*)
			
			(*Nodes States*)
			DiscreteNode_OK: BOOL;
			
			(*Cable Break Warning Flags*)
			ECatSlave_Cable_Breaks: UDINT;
			EP1918_NotPresent :BOOL;				(*Coupler is Not Present on Bus when expected*)
			EP1918_PortB_MissingLink: BOOL; 		
			EP1008_PortB_MissingLink: BOOL;			
			EP2624_PortB_MissingLink: BOOL;			
		
		(*CoE Read*)
			CoE_ReadFB_1: FB_EcCoESdoReadEx; 		(*FB to retrieve Data from terminals via CoE*)
			CoE_ReadBuffer_1: ARRAY [0..1] OF BYTE;	(*Variable, 2 bytes, for receiving data*)
			CoE_ReadErr_1: BOOL;					(*CoE Read Error Flag*)
			CoE_ReadErrID_1: UDINT;					(*CoE Read Error Identification*)
			CoE_ReadFB_2: FB_EcCoESdoReadEx; 		(*FB to retrieve Data from terminals via CoE*)
			CoE_ReadBuffer_2: ARRAY [0..1] OF BYTE;	(*Variable, 2 bytes, for receiving data*)
			CoE_ReadErr_2: BOOL;					(*CoE Read Error Flag*)
			CoE_ReadErrID_2: UDINT;					(*CoE Read Error Identification*)
			EP1918_Overtemperature: BOOL;			(*Flag for result of CoE Read*)
			
			(*DoorClosed_Safety_Switches: BOOL;*)	(*TLK MOVE TO INPUTS*)
			DoorClose_CMD: BOOL;
			DoorOpen_CMD: BOOL;
			DoorStop_CMD: BOOL;
			Door_CloseSR: SR;						(*Latch to Close the door*)
			Door_OpenSR: SR;						(*Latch to Open the door*)
			DoorOpened_TMR: TON;					(*Timer to say door is open, no door open switches*)
			DoorClosed_TMR: TON;					(*Timer to say door is closed*)
			DoorStop_TMR: TON;

	END_VAR

	VAR_OUTPUT
			
			(*Internal Output Variables*)
			FB_OK: BOOL;
			Discrete_Image: udt_MDxx_Image_20251008;

			Door_Closed: BOOL;						(*Door is closed*)
			Door_Opened: BOOL;						(*Door is open*)
			Door_Running: BOOL;						(*Door is Running Open/Close*)
			Door_Faulted: BOOL;						(*Door is Faulted*)
			Door_Stopped: BOOL;						(*Door is Faulted*)

	END_VAR

(*		
	- DEBUG, this FB must be proven and debugged in field!!!! THEN remove THIS comment, b.lekx-toniolo
*)


	(*Set FB_OK to True*)
	FB_OK:= TRUE;
	
(*$$$$$$$$$$$$$$$$$$$$$$$$$$$$$$$$$$$$$$$$$$$$$$$$Gather Status Of Hardware $$$$$$$$$$$$$$$$$$$$$$$$$$$$$$$$$$$$$$$$$$$$$$$$$$$$*)
	(*Discrete I/O Node*)
	IF N01_STAT.InfoData.State=8 AND N02.InfoData.State=8 AND N03_STAT.InfoData.State=8
		THEN DiscreteNode_OK:=TRUE;
	ELSE DiscreteNode_OK:=FALSE;
	END_IF;

	(*Develop Port Connection Warning Flags*)
	IF N01_STAT.InfoData.State=257  (*State Machine for Slave Not Present*)
		THEN EP1918_NotPresent:= TRUE;
	ELSE EP1918_NotPresent := FALSE;
	END_IF;

	IF N01_STAT.InfoData.State=9224 (*State Machine for Link Missing at Port B*)
		THEN EP1918_PortB_MissingLink:= TRUE; (*PortB is OUT Port*)
	ELSE EP1918_PortB_MissingLink := FALSE;
	END_IF;
	
	IF (N02.InfoData.State = 9224) (*State Machine for Link Missing at Port B*)
		THEN EP1008_PortB_MissingLink:= TRUE; 
	ELSE EP1008_PortB_MissingLink := FALSE;
	END_IF;

	IF (N03_STAT.InfoData.State = 9224) (*State Machine for Link Missing at Port B*)
		THEN EP2624_PortB_MissingLink:= TRUE; 
	ELSE EP2624_PortB_MissingLink := FALSE;
	END_IF;
	
	(*Wrap up break Flags to Variable for shipment to UI*)
	ECatSlave_Cable_Breaks.0:= EP1918_NotPresent AND Prev_EcatNode_Present;
	ECatSlave_Cable_Breaks.1:= EP1918_PortB_MissingLink;
	ECatSlave_Cable_Breaks.2:= EP1008_PortB_MissingLink;
	ECatSlave_Cable_Breaks.3:= EP2624_PortB_MissingLink;

(*------------ CoE Reads ------------*)

	(*Read EP1918 Primaray Temperature Data*)

	(*FB Inputs*)
	CoE_ReadFB_1.bExecute:= CoE_Read_Trigger
							AND (N01_Stat.InfoData.State=8);					(*Execute Upon Trigger*)
	CoE_ReadFB_1.sNetId:= Ecat_Master_AmsNetID;
	CoE_ReadFB_1.nSlaveAddr:= N01_STAT.InfoData.AdsAddr.port;					(*Address of Ecat Slave being Read*)
	CoE_ReadFB_1.nIndex:= 16#F984;												(*CANopen SDO Index of Object (F984 = Device Info Data C1)*)
	CoE_ReadFB_1.nSubIndex:= 16#02;												(*CANopen SDO SubIndex (Location from Index) of Object*)
	CoE_ReadFB_1.cbBufLen:= 2;													(*Limit on Receive Length (bytes)*)
	CoE_ReadFB_1.pDstBuf:= ADR(CoE_ReadBuffer_1);								(*Pointer to Receive Buffer*)
	CoE_ReadFB_1.tTimeout:= T#2s;												(*TImeout for Read*)
	CoE_ReadFB_1.bCompleteAccess:= TRUE;										(*Allow Complete Access to Full SDO Object*)

	(*Execute FB*)
	CoE_ReadFB_1();

	(*FB Outputs*)
	CoE_ReadErr_1:= CoE_ReadFB_1.bError;										(*Error Flag of Read*)
	CoE_ReadErrID_1:= CoE_ReadFB_1.nErrId;										(*Error ID of Read (See ADS Return Codes)*)

	(*Read EP1918 Secondary Temperature Data*)

	(*FB Inputs*)
	CoE_ReadFB_2.bExecute:= CoE_Read_Trigger
							AND (N01_Stat.InfoData.State=8);					(*Execute Upon Trigger*)
	CoE_ReadFB_2.sNetId:= Ecat_Master_AmsNetID;
	CoE_ReadFB_2.nSlaveAddr:= N01_STAT.InfoData.AdsAddr.port;					(*Address of Ecat Slave being Read*)
	CoE_ReadFB_2.nIndex:= 16#F985;												(*CANopen SDO Index of Object (F985 = Device Info Data C2)*)
	CoE_ReadFB_2.nSubIndex:= 16#02;												(*CANopen SDO SubIndex (Location from Index) of Object*)
	CoE_ReadFB_2.cbBufLen:= 2;													(*Limit on Receive Length (bytes)*)
	CoE_ReadFB_2.pDstBuf:= ADR(CoE_ReadBuffer_2);								(*Pointer to Receive Buffer*)
	CoE_ReadFB_2.tTimeout:= T#2S;												(*TImeout for Read*)
	CoE_ReadFB_2.bCompleteAccess:= TRUE;										(*Allow Complete Access to Full SDO Object*)

	(*Execute FB*)
	CoE_ReadFB_2();

	(*FB Outputs*)
	CoE_ReadErr_2:= CoE_ReadFB_2.bError;										(*Error Flag of Read*)
	CoE_ReadErrID_2:= CoE_ReadFB_2.nErrId;										(*Error ID of Read (See ADS Return Codes)*)
	
	
	
	
	(*Tranfer Data to Image*)
	IF (N01_Stat.InfoData.State=8) AND NOT CoE_ReadErr_1 AND NOT CoE_ReadErr_2
		THEN
		N01_STAT.CoE_Temperature_1:= FUN_GTAC_BYTEStoINT(CoE_ReadBuffer_1[0],CoE_ReadBuffer_1[1]);	(*Grab bytes 0 and 1 of read buffer, this is Primary Temperature*)
		N01_STAT.CoE_Temperature_2:= FUN_GTAC_BYTEStoINT(CoE_ReadBuffer_1[0],CoE_ReadBuffer_1[1]);	(*Grab bytes 0 and 1 of read buffer, this is Secondary Temperature*)
	ELSE
		(*If Read Error, then blank data*)
		N01_STAT.CoE_Temperature_1:=0;
		N01_STAT.CoE_Temperature_2:=0;
	END_IF;

	(*Finally Evaluate Temperature Vs Upper Limit Restrictions*)
	IF (N01_STAT.CoE_Temperature_1>=90) OR (N01_STAT.CoE_Temperature_2>=90)
		THEN
		EP1918_Overtemperature:= TRUE;
	ELSE
		EP1918_Overtemperature:= FALSE;
	END_IF;
	
	

(*$$$$$$$$$$$$$$$$$$$$$$$$$$$$$$$$$$$$$$$$$$$$$ Gather Safety Inputs $$$$$$$$$$$$$$$$$$$$$$$$$$$$$$$$$$$$$$$$$$$$$$$$$$$$$$$$$*)
	(*Door Safety Switches*)
	(*DoorClosed_Safety_Switches:= N01_STAT.I.0 AND N01_STAT.I.1 AND N01_STAT.I.2 AND N01_STAT.I.3;*)


(*$$$$$$$$$$$$$$$$$$$$$$$$$$$$$$$$$$$$$$$$$$$$ Gather Standard Inputs $$$$$$$$$$$$$$$$$$$$$$$$$$$$$$$$$$$$$$$$$$$$$$$$$$$$$$$$*)

	Door_Closed:= 	N02.I.0 AND DoorClosed_Safety_Switches;		(*YDC0*)
	Door_Opened:= 	N02.I.1;									(*YDC1*)
	Door_Stopped:= 	N02.I.2;									(*YDC2*)
	Door_Faulted:= 	N02.I.3;									(*YDC3*)
	
(*$$$$$$$$$$$$$$$$$$$$$$$$$$$$$$$$$$$$$$$$$$$$$ Internal Code $$$$$$$$$$$$$$$$$$$$$$$$$$$$$$$$$$$$$$$$$$$$$$$$$$$$$$$$$*)

	(*Set Door to Close*)
	Door_CloseSR(
			SET1:= Enable_Motion AND Enable_Latch AND DoorClose_REQ AND NOT DoorOpen_REQ,
			RESET:= NOT Enable_Motion OR NOT Enable_Latch OR DoorOpen_REQ OR Door_Closed,
			Q1=>
			);

	(*Set Door to Open*)
	Door_OpenSR(
			SET1:= Enable_Latch AND DoorOpen_REQ AND NOT DoorClose_REQ,
			RESET:= NOT Enable_Latch OR DoorClose_REQ OR Door_Opened,
			Q1=>
			);

	(*Output to Open or Close the Door*)
	DoorClose_CMD:= Enable_Motion AND ((Enable_Latch AND Door_CloseSR.Q1) OR (NOT Enable_Latch AND DoorClose_REQ)) AND NOT Door_OpenSR.Q1;
	DoorOpen_CMD:= ((Enable_Latch AND Door_OpenSR.Q1) OR (NOT Enable_Latch AND DoorOpen_REQ)) AND NOT Door_CloseSR.Q1;
	DoorStop_CMD:= DoorStop_REQ AND (NOT Door_Closed OR NOT Door_Opened);

	(*Door Opened Timer*)
	DoorOpened_TMR(
			IN:= NOT DoorClosed_Safety_Switches AND DoorOpen_CMD,
			PT:= T#2.75s,
			Q=> ,
			ET=>
			);

	(*Door Closed Timer*)
	DoorClosed_TMR(
			IN:= DoorClosed_Safety_Switches,
			PT:= T#500ms,
			Q=> ,
			ET=>
			);
			
		(*Door Stop Timer*)
	DoorStop_TMR(
			IN:= DoorStop_REQ,
			PT:= T#200MS,
			Q=> ,
			ET=>
			);
			
(*$$$$$$$$$$$$$$$$$$$$$$$$$$$$$$$$$$$$$$$$$$$$$$$$$$$ Faults $$$$$$$$$$$$$$$$$$$$$$$$$$$$$$$$$$$$$$$$$$$$$$$$$$$$$$$*)


(*$$$$$$$$$$$$$$$$$$$$$$$$$$$$$$$$$$$$$$$$$$$$$$ Transfer Standard Outputs $$$$$$$$$$$$$$$$$$$$$$$$$$$$$$$$$$$$$$$$$$$*)
	(*Transfer I/O Images for Display On HMI*)
	Discrete_Image.N01_STAT:= N01_STAT;
	Discrete_Image.N02:= N02;
	Discrete_Image.N03:= N03;
	Discrete_Image.N03_STAT:= N03_STAT;

(*Transfer Commands to Discrete Node Outputs*)
	N03.Q.0:= DoorOpen_CMD;	     	(*X2*)
	N03.Q.1:= DoorClose_CMD;		(*X5*)
	N03.Q.2:= DoorStop_CMD;				(*X6*)
	N03.Q.3:= FALSE;				(*X7*)
	N03.Q.4:= (*DoorStop_CMD*) FALSE;			(*X8*)
	N03.Q.5:= FALSE;				(*X9*)
	N03.Q.6:= FALSE;				(*X10*)
	N03.Q.7:= FALSE;				(*X11*)


(*$$$$$$$$$$$$$$$$$$$$$$$$$$$$$$$$$$$$$$$$$$$$$$ Transfer Safety Outputs $$$$$$$$$$$$$$$$$$$$$$$$$$$$$$$$$$$$$$$$$$$*)

	(*Set All Safety Groups to Run*)
		N01_CMD.SGs_RUNSTOP:= TRUE;
	(*Reset Of Safety Group Errors*)
		N01_CMD.SGs_ERRAck:= Safety_RST;
	(*Reset Only Used FBs With In Safety Group*)
		(*Reset of Estop, Safety Gate and Misc FBs*)
		N01_CMD.FBs_ControlPowerPB:= Safety_RST;
		(*Retrigger of evaluation of Switches*)
		N01_CMD.FBs_Restart_Spare:= OPxx_RST;

END_FUNCTION_BLOCK

// ---- POUs/FBs/FB_GTAC_Conveyor_20210303.TcPOU
(*FB for use with Conveyors

	Original Author(s): Justin Vandongen of Sodecia GTAC.; 
------------------------------------------------------------------------------------------
REVISION NOTES:
	Version 20201013
		- intial concept, J.Vandongen
	Version 20210303
		- added timeout functionality, j.underhill
------------------------------------------------------------------------------------------
*)


FUNCTION_BLOCK FB_GTAC_Conveyor_20210303
	VAR_INPUT
		Enable_Motion: BOOL;
		Enable_Start_Latch: BOOL;
		Reset_TimeOut: BOOL;

		Start_Delay_Time: TIME;
		Stop_Delay_Time: TIME;
		TimeOut_Time: TIME;

		Start_Conveyor: BOOL;
		Pause_Conveyor: BOOL;
		Stop_Conveyor: BOOL;
	
	
	END_VAR


	VAR
		Start_Latch: SR;
		Stop_Latch: SR;

		Start_DelayTMR: TON;
		Stop_DelayTMR: TON;
		TimeOutTMR: TON;


	END_VAR
	

	VAR_OUTPUT
		FB_OK: BOOL;
		Conveyor_On_CMD: BOOL;


	END_VAR

	(*Set FB_OK to True*)
	FB_OK:= TRUE;


(*$$$$$$$$$$$$$$$$$$$$$$$$$$$$$$$$$$$$$$$$$$$$$$$$$$ Internal Code $$$$$$$$$$$$$$$$$$$$$$$$$$$$$$$$$$$$$$$$$$$$$$$$$$$$$$$$*)

	(*Start Latch to keep conveyor on until stop signal is present*)
	Start_Latch(
			SET1:= Enable_Start_Latch AND Start_Conveyor
					AND NOT Stop_Conveyor AND NOT Pause_Conveyor AND NOT TimeOutTMR.Q,
			RESET:= Stop_Conveyor AND Stop_DelayTMR.Q,
			Q1=> );

	(*Capture Stop Conditions*)
	Stop_Latch(
			Set1:= Stop_Conveyor OR Pause_Conveyor,
			RESET:= Stop_DelayTMR.Q,
			Q1=> );

	(*Timer used to timeout conveyor after running for X time*)
	TimeOutTMR(
				IN:= (Conveyor_On_CMD OR TimeOutTMR.Q) AND NOT Reset_TimeOut,
				PT:= TimeOut_Time,
				Q=> ,
				ET=> );


	(*Timer used to delay the start of the conveyor until it sees the Start_Conveyor signal for a duration of time first*)
	Start_DelayTMR(
			IN:= Enable_Motion AND (Start_Conveyor OR Start_Latch.Q1),
			PT:= Start_Delay_Time,
			Q=> ,
			ET=> );


	(*Timer used to keep the conveyor running after the stop signal has been turned on. Ideally used to control the stop position*)
	Stop_DelayTMR(
			IN:= Enable_Motion AND Stop_Latch.Q1,
			PT:= Stop_Delay_Time,
			Q=> ,
			ET=> );


(*$$$$$$$$$$$$$$$$$$$$$$$$$$$$$$$$$$$$$$$$$$$$$$ Transfer Standard Outputs $$$$$$$$$$$$$$$$$$$$$$$$$$$$$$$$$$$$$$$$$$$*)


	Conveyor_On_CMD:= Enable_Motion
				AND ((Start_Conveyor OR Start_Latch.Q1) AND Start_DelayTMR.Q);




(*end*)

END_FUNCTION_BLOCK

// ---- POUs/FBs/FB_SCHNEIDERVFD_20180808.TcPOU
(*FB for use with Schenider Electric VFD:
	Original Author(s): Justin Vandongen of Sodecia GTAC; 
------------------------------------------------------------------------------------------
REVISION NOTES:
	Version 20180808
		- Initial Concept, j.vandongen
		- max output frequency is setup to 50hz. in future projects this could change and scalling will need to change. j.vandongen

------------------------------------------------------------------------------------------
*)




FUNCTION_BLOCK FB_SchneiderVFD_20180808

	VAR_INPUT
		Enable_Motion: BOOL;
		All_Safeties_OK: BOOL;
		Prev_EcatNode_Present: BOOL;

		(*Control Word*)
		Operating_State_Switch_On: BOOL; 			(*Bit 0*)
		Enable_Voltage: BOOL;					(*Bit 1*)
		Operating_State_Quick_Stop_Req: BOOL; 	(*Bit 2*)
		Enable_Operation: BOOL;					(*Bit 3*)
		Operating_Mode_Bit4: BOOL;				(*Bit 4*)
		Operating_Mode_Bit5: BOOL;				(*Bit 5*)
		Operating_Mode_Bit6: BOOL;				(*Bit 6*)
		Fault_Reset: BOOL;						(*Bit 7*)
		Halt: BOOL;								(*Bit 8*)
		Operating_Mode_Bit9: BOOL;				(*Bit 9*)

		Requested_Freq: UINT;

	END_VAR


	VAR
	(*Inputs from VFD*)
		Status_Word AT %I*: UINT;

	(*Outputs to VFD*)
		Control_Word AT %Q*: UINT;
		Target_Velocity AT %Q*: INT;

	(*Hardware Data Types*)
		VFD_State AT %I*: udt_Schneider_VFD_20180808;

	(* Nodes/Interface States*)
		DiscreteNode_OK: BOOL;

	(*Cable Break Warning Flags*)
		ECatSlave_Cable_Breaks: UDINT;
		ATV320_NotPresent :BOOL;			(*Bridge Terminal is not on Bus when expected*)
		ATV320_PortB_MissingLink: BOOL;

		(*Move time*)
		Move_TMR: TON;

		Test: UINT;


	END_VAR


	VAR_OUTPUT
		FB_OK: BOOL;

	(*Status_Word*)
		Operating_State_Ready: BOOL;					(*Bit 0*)
		Operating_State_Switched_On: BOOL;			(*Bit 1*)
		Operating_State_Operation_enabled: BOOL;		(*Bit 2*)
		Operating_State_Fault: BOOL;					(*Bit 3*)
		Voltage_Enabled: BOOL;						(*Bit 4*)
		Operating_State_Quick_Stop: BOOL;				(*Bit 5*)
		Operating_State_Switch_On_Dissabled: BOOL;	(*Bit 6*)
		Error_Class0: BOOL;							(*Bit 7*)
		Halt_Requested: BOOL;						(*Bit 8*)
		Remote: BOOL;								(*Bit 9*)
		Target_Reached: BOOL;						(*Bit 10*)
		Internal_Limit: BOOL;							(*Bit 11*)
		Operating_Mode_Specific: BOOL;				(*Bit 12*)
		X_ERR: BOOL;								(*Bit 13*)
		X_End: BOOL;								(*Bit 14*)
		Ref_OK: BOOL;								(*Bit 15*)

		Faulted: BOOL;
		Move_TIME: TIME;

		Discrete_Image: udt_Schneider_VFD_Image_20180808;

	END_VAR

	(*Set FB_OK to True*)
		FB_OK:= TRUE;

(*$$$$$$$$$$$$$$$$$$$$$$$$$$$$$$$$$$$$$$$$$$$$$$$$Gather Status Of Hardware $$$$$$$$$$$$$$$$$$$$$$$$$$$$$$$$$$$$$$$$$$$$$$$$$$$$*)

		IF (VFD_State.InfoData.State=8)
			THEN DiscreteNode_OK:= TRUE;
		ELSE DiscreteNode_OK:= FALSE;
		END_IF;

		(*Develop Port Connection Warning Flags*)
		IF (VFD_STATE.InfoData.State=257) (*State Machine for Slave Not Present*)
			THEN ATV320_NotPresent:= TRUE;
		ELSE ATV320_NotPresent := FALSE;
		END_IF;

		IF (VFD_STATE.InfoData.State= 9224) (*State Machine for Link Missing at Port B*)
			THEN ATV320_PortB_MissingLink:= TRUE; (*PortB is OUT Port*)
		ELSE ATV320_PortB_MissingLink := FALSE;
		END_IF;

